LIN {X 0,Y 419.941,Z 601.82,A -85,B 0,C 180,E1 -10275.874,E2 -10275.874} C_VEL
LIN {X 0,Y 423.055,Z 612.363,A -85,B 0,C 180,E1 -10276.249,E2 -10276.249} C_VEL
LIN {X 0,Y 424.407,Z 618.673,A -85,B 0,C 180,E1 -10276.443,E2 -10276.443} C_VEL
LIN {X 0,Y 422.961,Z 707.954,A -85,B 0,C 180,E1 -10278.121,E2 -10278.121} C_VEL
LIN {X 0,Y 422.595,Z 721.713,A -85,B 0,C 180,E1 -10278.586,E2 -10278.586} C_VEL
LIN {X 0,Y 422.096,Z 733.741,A -85,B 0,C 180,E1 -10279.179,E2 -10279.179} C_VEL
LIN {X 0,Y 421.512,Z 745.803,A -85,B 0,C 180,E1 -10279.987,E2 -10279.987} C_VEL
LIN {X 0,Y 420.851,Z 757.025,A -85,B 0,C 180,E1 -10280.949,E2 -10280.949} C_VEL
LIN {X 0,Y 420.101,Z 766.764,A -85,B 0,C 180,E1 -10281.982,E2 -10281.982} C_VEL
LIN {X 0,Y 419.384,Z 776.447,A -85,B 0,C 180,E1 -10283.26,E2 -10283.26} C_VEL
LIN {X 0,Y 418.78,Z 784.344,A -85,B 0,C 180,E1 -10284.542,E2 -10284.542} C_VEL
LIN {X 0,Y 418.327,Z 791.168,A -85,B 0,C 180,E1 -10285.9,E2 -10285.9} C_VEL
LIN {X 0,Y 417.852,Z 797.772,A -85,B 0,C 180,E1 -10287.55,E2 -10287.55} C_VEL
LIN {X 0,Y 417.506,Z 802.788,A -85,B 0,C 180,E1 -10289.22,E2 -10289.22} C_VEL
LIN {X 0,Y 417.277,Z 806.247,A -85,B 0,C 180,E1 -10290.802,E2 -10290.802} C_VEL
LIN {X 0,Y 417.079,Z 808.819,A -85,B 0,C 180,E1 -10292.63,E2 -10292.63} C_VEL
LIN {X 0,Y 416.972,Z 809.86,A -85,B 0,C 180,E1 -10294.324,E2 -10294.324} C_VEL
LIN {X 0,Y 417.022,Z 809.583,A -85,B 0,C 180,E1 -10296.146,E2 -10296.146} C_VEL
LIN {X 0,Y 417.033,Z 808.324,A -85,B 0,C 180,E1 -10297.624,E2 -10297.624} C_VEL
LIN {X 0,Y 417.228,Z 805.887,A -85,B 0,C 180,E1 -10299.211,E2 -10299.211} C_VEL
LIN {X 0,Y 417.434,Z 802.41,A -85,B 0,C 180,E1 -10300.747,E2 -10300.747} C_VEL
LIN {X 0,Y 417.657,Z 797.653,A -85,B 0,C 180,E1 -10302.306,E2 -10302.306} C_VEL
LIN {X 0,Y 418.108,Z 791.143,A -85,B 0,C 180,E1 -10303.936,E2 -10303.936} C_VEL
LIN {X 0,Y 418.574,Z 784.013,A -85,B 0,C 180,E1 -10305.349,E2 -10305.349} C_VEL
LIN {X 0,Y 419.196,Z 775.516,A -85,B 0,C 180,E1 -10306.712,E2 -10306.712} C_VEL
LIN {X 0,Y 419.844,Z 765.863,A -85,B 0,C 180,E1 -10307.967,E2 -10307.967} C_VEL
LIN {X 0,Y 420.512,Z 755.212,A -85,B 0,C 180,E1 -10309.076,E2 -10309.076} C_VEL
LIN {X 0,Y 421.141,Z 744.253,A -85,B 0,C 180,E1 -10309.991,E2 -10309.991} C_VEL
LIN {X 0,Y 421.739,Z 733.285,A -85,B 0,C 180,E1 -10310.712,E2 -10310.712} C_VEL
LIN {X 0,Y 422.186,Z 720.348,A -85,B 0,C 180,E1 -10311.348,E2 -10311.348} C_VEL
LIN {X 0,Y 422.524,Z 707.087,A -85,B 0,C 180,E1 -10311.789,E2 -10311.789} C_VEL
LIN {X 0,Y 423.711,Z 617.543,A -85,B 0,C 180,E1 -10313.442,E2 -10313.442} C_VEL
LIN {X 0,Y 420.089,Z 601.796,A -85,B 0,C 180,E1 -10313.898,E2 -10313.898} C_VEL
LIN {X 0,Y 419.451,Z 599.695,A -85,B 0,C 180,E1 -10313.985,E2 -10313.985} C_VEL
LIN {X 0,Y 418.293,Z 593.383,A -85,B 0,C 180,E1 -10315.671,E2 -10315.671} C_VEL
LIN {X 0,Y 418.23,Z 593.385,A -85,B 0,C 180,E1 -10319.157,E2 -10319.157} C_VEL
LIN {X 0,Y 418.288,Z 593.383,A -85,B 0,C 180,E1 -10321.938,E2 -10321.938} C_VEL
LIN {X 0,Y 418.276,Z 593.378,A -85,B 0,C 180,E1 -10323.348,E2 -10323.348} C_VEL
LIN {X 0,Y 417.581,Z 593.471,A -85,B 0,C 180,E1 -10324.151,E2 -10324.151} C_VEL
LIN {X 0,Y 414.714,Z 593.823,A -85,B 0,C 180,E1 -10325.457,E2 -10325.457} C_VEL
LIN {X 0,Y 412.306,Z 594.125,A -85,B 0,C 180,E1 -10326.511,E2 -10326.511} C_VEL
LIN {X 0,Y 411.279,Z 594.25,A -85,B 0,C 180,E1 -10327.325,E2 -10327.325} C_VEL
LIN {X 0,Y 411.198,Z 594.261,A -85,B 0,C 180,E1 -10327.601,E2 -10327.601} C_VEL
LIN {X 0,Y 411.234,Z 594.255,A -85,B 0,C 180,E1 -10331.053,E2 -10331.053} C_VEL
LIN {X 0,Y 411.254,Z 594.259,A -85,B 0,C 180,E1 -10334.133,E2 -10334.133} C_VEL
LIN {X 0,Y 411.314,Z 594.245,A -85,B 0,C 180,E1 -10337.167,E2 -10337.167} C_VEL
LIN {X 0,Y 411.308,Z 594.251,A -85,B 0,C 180,E1 -10340.163,E2 -10340.163} C_VEL
LIN {X 0,Y 411.461,Z 594.228,A -85,B 0,C 180,E1 -10343.134,E2 -10343.134} C_VEL
LIN {X 0,Y 411.312,Z 594.247,A -85,B 0,C 180,E1 -10345.1,E2 -10345.1} C_VEL
LIN {X 0,Y 411.515,Z 594.222,A -85,B 0,C 180,E1 -10348.044,E2 -10348.044} C_VEL
LIN {X 0,Y 411.642,Z 594.206,A -85,B 0,C 180,E1 -10350.001,E2 -10350.001} C_VEL
LIN {X 0,Y 411.468,Z 594.23,A -85,B 0,C 180,E1 -10352.938,E2 -10352.938} C_VEL
LIN {X 0,Y 411.463,Z 594.232,A -85,B 0,C 180,E1 -10356.868,E2 -10356.868} C_VEL
LIN {X 0,Y 411.296,Z 594.248,A -85,B 0,C 180,E1 -10359.84,E2 -10359.84} C_VEL
LIN {X 0,Y 411.308,Z 594.25,A -85,B 0,C 180,E1 -10363.105,E2 -10363.105} C_VEL
LIN {X 0,Y 411.266,Z 594.259,A -85,B 0,C 180,E1 -10366.87,E2 -10366.87} C_VEL
LIN {X 0,Y 411.234,Z 594.255,A -85,B 0,C 180,E1 -10369.988,E2 -10369.988} C_VEL
LIN {X 0,Y 411.206,Z 594.264,A -85,B 0,C 180,E1 -10373.148,E2 -10373.148} C_VEL
LIN {X 0,Y 411.241,Z 594.255,A -85,B 0,C 180,E1 -10376.382,E2 -10376.382} C_VEL
LIN {X 0,Y 411.204,Z 594.26,A -85,B 0,C 180,E1 -10379.713,E2 -10379.713} C_VEL
LIN {X 0,Y 411.21,Z 594.266,A -85,B 0,C 180,E1 -10383.156,E2 -10383.156} C_VEL
LIN {X 0,Y 411.197,Z 594.261,A -85,B 0,C 180,E1 -10386.553,E2 -10386.553} C_VEL
LIN {X 0,Y 411.219,Z 594.26,A -85,B 0,C 180,E1 -10389.729,E2 -10389.729} C_VEL
LIN {X 0,Y 411.177,Z 594.268,A -85,B 0,C 180,E1 -10393.134,E2 -10393.134} C_VEL
LIN {X 0,Y 411.172,Z 594.265,A -85,B 0,C 180,E1 -10395.882,E2 -10395.882} C_VEL
LIN {X 0,Y 411.167,Z 594.264,A -85,B 0,C 180,E1 -10398.772,E2 -10398.772} C_VEL
LIN {X 0,Y 411.196,Z 594.262,A -85,B 0,C 180,E1 -10402.027,E2 -10402.027} C_VEL
LIN {X 0,Y 411.211,Z 594.265,A -85,B 0,C 180,E1 -10405.667,E2 -10405.667} C_VEL
LIN {X 0,Y 411.194,Z 594.262,A -85,B 0,C 180,E1 -10409.153,E2 -10409.153} C_VEL
LIN {X 0,Y 411.264,Z 594.252,A -85,B 0,C 180,E1 -10412.523,E2 -10412.523} C_VEL
LIN {X 0,Y 411.225,Z 594.264,A -85,B 0,C 180,E1 -10415.785,E2 -10415.785} C_VEL
LIN {X 0,Y 411.201,Z 594.26,A -85,B 0,C 180,E1 -10418.966,E2 -10418.966} C_VEL
LIN {X 0,Y 411.256,Z 594.257,A -85,B 0,C 180,E1 -10422.085,E2 -10422.085} C_VEL
LIN {X 0,Y 411.265,Z 594.252,A -85,B 0,C 180,E1 -10425.148,E2 -10425.148} C_VEL
LIN {X 0,Y 411.288,Z 594.254,A -85,B 0,C 180,E1 -10428.168,E2 -10428.168} C_VEL
LIN {X 0,Y 411.446,Z 594.235,A -85,B 0,C 180,E1 -10432.189,E2 -10432.189} C_VEL
LIN {X 0,Y 411.477,Z 594.232,A -85,B 0,C 180,E1 -10434.118,E2 -10434.118} C_VEL
LIN {X 0,Y 411.517,Z 594.226,A -85,B 0,C 180,E1 -10438.043,E2 -10438.043} C_VEL
LIN {X 0,Y 411.646,Z 594.209,A -85,B 0,C 180,E1 -10440,E2 -10440} C_VEL
LIN {X 0,Y 411.463,Z 594.227,A -85,B 0,C 180,E1 -10442.937,E2 -10442.937} C_VEL
LIN {X 0,Y 411.462,Z 594.229,A -85,B 0,C 180,E1 -10446.867,E2 -10446.867} C_VEL
LIN {X 0,Y 411.298,Z 594.249,A -85,B 0,C 180,E1 -10449.839,E2 -10449.839} C_VEL
LIN {X 0,Y 411.311,Z 594.246,A -85,B 0,C 180,E1 -10453.104,E2 -10453.104} C_VEL
LIN {X 0,Y 411.263,Z 594.255,A -85,B 0,C 180,E1 -10456.889,E2 -10456.889} C_VEL
LIN {X 0,Y 411.236,Z 594.256,A -85,B 0,C 180,E1 -10459.987,E2 -10459.987} C_VEL
LIN {X 0,Y 411.202,Z 594.261,A -85,B 0,C 180,E1 -10463.148,E2 -10463.148} C_VEL
LIN {X 0,Y 411.243,Z 594.258,A -85,B 0,C 180,E1 -10466.381,E2 -10466.381} C_VEL
LIN {X 0,Y 411.206,Z 594.259,A -85,B 0,C 180,E1 -10469.712,E2 -10469.712} C_VEL
LIN {X 0,Y 411.212,Z 594.261,A -85,B 0,C 180,E1 -10473.156,E2 -10473.156} C_VEL
LIN {X 0,Y 411.198,Z 594.264,A -85,B 0,C 180,E1 -10476.552,E2 -10476.552} C_VEL
LIN {X 0,Y 411.216,Z 594.258,A -85,B 0,C 180,E1 -10479.727,E2 -10479.727} C_VEL
LIN {X 0,Y 411.179,Z 594.268,A -85,B 0,C 180,E1 -10483.133,E2 -10483.133} C_VEL
LIN {X 0,Y 411.173,Z 594.263,A -85,B 0,C 180,E1 -10485.881,E2 -10485.881} C_VEL
LIN {X 0,Y 411.169,Z 594.267,A -85,B 0,C 180,E1 -10488.771,E2 -10488.771} C_VEL
LIN {X 0,Y 411.21,Z 594.259,A -85,B 0,C 180,E1 -10491.831,E2 -10491.831} C_VEL
LIN {X 0,Y 411.216,Z 594.264,A -85,B 0,C 180,E1 -10495.121,E2 -10495.121} C_VEL
LIN {X 0,Y 411.171,Z 594.266,A -85,B 0,C 180,E1 -10498.002,E2 -10498.002} C_VEL
LIN {X 0,Y 411.261,Z 594.413,A -85,B 0,C 180,E1 -10500.79,E2 -10500.79} C_VEL
LIN {X 0,Y 414.087,Z 607.419,A -85,B 0,C 180,E1 -10503.542,E2 -10503.542} C_VEL
LIN {X 0,Y 414.89,Z 613.069,A -85,B 0,C 180,E1 -10504.687,E2 -10504.687} C_VEL
LIN {X 0,Y 413.836,Z 628.092,A -85,B 0,C 180,E1 -10507.535,E2 -10507.535} C_VEL
LIN {X 0,Y 412.832,Z 643.304,A -85,B 0,C 180,E1 -10510.378,E2 -10510.378} C_VEL
LIN {X 0,Y 412.697,Z 645.191,A -85,B 0,C 180,E1 -10510.729,E2 -10510.729} C_VEL
LIN {X 0,Y 416.641,Z 674.102,A -85,B 0,C 180,E1 -10511.462,E2 -10511.462} C_VEL
LIN {X 0,Y 415.489,Z 754.532,A -85,B 0,C 180,E1 -10512.971,E2 -10512.971} C_VEL
LIN {X 0,Y 414.975,Z 768.128,A -85,B 0,C 180,E1 -10513.424,E2 -10513.424} C_VEL
LIN {X 0,Y 414.351,Z 779.945,A -85,B 0,C 180,E1 -10514,E2 -10514} C_VEL
LIN {X 0,Y 413.654,Z 791.204,A -85,B 0,C 180,E1 -10514.73,E2 -10514.73} C_VEL
LIN {X 0,Y 412.918,Z 802.904,A -85,B 0,C 180,E1 -10515.712,E2 -10515.712} C_VEL
LIN {X 0,Y 412.199,Z 813.634,A -85,B 0,C 180,E1 -10516.839,E2 -10516.839} C_VEL
LIN {X 0,Y 411.651,Z 822.069,A -85,B 0,C 180,E1 -10517.927,E2 -10517.927} C_VEL
LIN {X 0,Y 411.016,Z 830.01,A -85,B 0,C 180,E1 -10519.158,E2 -10519.158} C_VEL
LIN {X 0,Y 410.584,Z 837.764,A -85,B 0,C 180,E1 -10520.64,E2 -10520.64} C_VEL
LIN {X 0,Y 410.274,Z 843.987,A -85,B 0,C 180,E1 -10522.122,E2 -10522.122} C_VEL
LIN {X 0,Y 410.107,Z 849.181,A -85,B 0,C 180,E1 -10523.695,E2 -10523.695} C_VEL
LIN {X 0,Y 410.079,Z 852.686,A -85,B 0,C 180,E1 -10525.083,E2 -10525.083} C_VEL
LIN {X 0,Y 409.971,Z 854.618,A -85,B 0,C 180,E1 -10526.067,E2 -10526.067} C_VEL
LIN {X 0,Y 410.053,Z 856.108,A -85,B 0,C 180,E1 -10527.052,E2 -10527.052} C_VEL
LIN {X 0,Y 410.059,Z 857.14,A -85,B 0,C 180,E1 -10528.035,E2 -10528.035} C_VEL
LIN {X 0,Y 410.027,Z 857.768,A -85,B 0,C 180,E1 -10529.017,E2 -10529.017} C_VEL
LIN {X 0,Y 410.033,Z 857.996,A -85,B 0,C 180,E1 -10529.999,E2 -10529.999} C_VEL
LIN {X 0,Y 410.027,Z 857.792,A -85,B 0,C 180,E1 -10530.981,E2 -10530.981} C_VEL
LIN {X 0,Y 410.06,Z 857.161,A -85,B 0,C 180,E1 -10531.963,E2 -10531.963} C_VEL
LIN {X 0,Y 410.055,Z 856.128,A -85,B 0,C 180,E1 -10532.946,E2 -10532.946} C_VEL
LIN {X 0,Y 409.969,Z 854.68,A -85,B 0,C 180,E1 -10533.931,E2 -10533.931} C_VEL
LIN {X 0,Y 410.042,Z 851.651,A -85,B 0,C 180,E1 -10535.408,E2 -10535.408} C_VEL
LIN {X 0,Y 410.163,Z 847.56,A -85,B 0,C 180,E1 -10536.888,E2 -10536.888} C_VEL
LIN {X 0,Y 410.411,Z 841.281,A -85,B 0,C 180,E1 -10538.616,E2 -10538.616} C_VEL
LIN {X 0,Y 410.816,Z 834.425,A -85,B 0,C 180,E1 -10540.098,E2 -10540.098} C_VEL
LIN {X 0,Y 411.389,Z 825.935,A -85,B 0,C 180,E1 -10541.579,E2 -10541.579} C_VEL
LIN {X 0,Y 411.949,Z 817.225,A -85,B 0,C 180,E1 -10542.813,E2 -10542.813} C_VEL
LIN {X 0,Y 412.72,Z 806.761,A -85,B 0,C 180,E1 -10544.017,E2 -10544.017} C_VEL
LIN {X 0,Y 413.498,Z 795.956,A -85,B 0,C 180,E1 -10545.021,E2 -10545.021} C_VEL
LIN {X 0,Y 414.343,Z 784.371,A -85,B 0,C 180,E1 -10545.872,E2 -10545.872} C_VEL
LIN {X 0,Y 415.045,Z 771.148,A -85,B 0,C 180,E1 -10546.602,E2 -10546.602} C_VEL
LIN {X 0,Y 415.738,Z 757.929,A -85,B 0,C 180,E1 -10547.111,E2 -10547.111} C_VEL
LIN {X 0,Y 416.035,Z 743.572,A -85,B 0,C 180,E1 -10547.447,E2 -10547.447} C_VEL
LIN {X 0,Y 417.035,Z 672.509,A -85,B 0,C 180,E1 -10548.788,E2 -10548.788} C_VEL
LIN {X 0,Y 413.245,Z 645.793,A -85,B 0,C 180,E1 -10549.525,E2 -10549.525} C_VEL
LIN {X 0,Y 412.815,Z 643.284,A -85,B 0,C 180,E1 -10549.621,E2 -10549.621} C_VEL
LIN {X 0,Y 414.034,Z 625.579,A -85,B 0,C 180,E1 -10552.979,E2 -10552.979} C_VEL
LIN {X 0,Y 414.946,Z 612.192,A -85,B 0,C 180,E1 -10555.573,E2 -10555.573} C_VEL
LIN {X 0,Y 413.027,Z 602.03,A -85,B 0,C 180,E1 -10557.77,E2 -10557.77} C_VEL
LIN {X 0,Y 411.226,Z 594.263,A -85,B 0,C 180,E1 -10559.539,E2 -10559.539} C_VEL
LIN {X 0,Y 411.203,Z 594.266,A -85,B 0,C 180,E1 -10563.155,E2 -10563.155} C_VEL
LIN {X 0,Y 411.193,Z 594.268,A -85,B 0,C 180,E1 -10566.552,E2 -10566.552} C_VEL
LIN {X 0,Y 411.224,Z 594.262,A -85,B 0,C 180,E1 -10569.729,E2 -10569.729} C_VEL
LIN {X 0,Y 411.173,Z 594.269,A -85,B 0,C 180,E1 -10573.132,E2 -10573.132} C_VEL
LIN {X 0,Y 411.231,Z 594.261,A -85,B 0,C 180,E1 -10575.87,E2 -10575.87} C_VEL
LIN {X 0,Y 411.205,Z 594.263,A -85,B 0,C 180,E1 -10578.763,E2 -10578.763} C_VEL
LIN {X 0,Y 411.199,Z 594.263,A -85,B 0,C 180,E1 -10582.027,E2 -10582.027} C_VEL
LIN {X 0,Y 411.2,Z 594.261,A -85,B 0,C 180,E1 -10585.666,E2 -10585.666} C_VEL
LIN {X 0,Y 411.194,Z 594.261,A -85,B 0,C 180,E1 -10589.153,E2 -10589.153} C_VEL
LIN {X 0,Y 411.252,Z 594.258,A -85,B 0,C 180,E1 -10592.522,E2 -10592.522} C_VEL
LIN {X 0,Y 411.219,Z 594.259,A -85,B 0,C 180,E1 -10595.784,E2 -10595.784} C_VEL
LIN {X 0,Y 411.189,Z 594.261,A -85,B 0,C 180,E1 -10598.965,E2 -10598.965} C_VEL
LIN {X 0,Y 411.245,Z 594.259,A -85,B 0,C 180,E1 -10602.084,E2 -10602.084} C_VEL
LIN {X 0,Y 411.254,Z 594.253,A -85,B 0,C 180,E1 -10605.147,E2 -10605.147} C_VEL
LIN {X 0,Y 411.291,Z 594.252,A -85,B 0,C 180,E1 -10608.167,E2 -10608.167} C_VEL
LIN {X 0,Y 411.473,Z 594.232,A -85,B 0,C 180,E1 -10612.146,E2 -10612.146} C_VEL
LIN {X 0,Y 411.467,Z 594.233,A -85,B 0,C 180,E1 -10614.118,E2 -10614.118} C_VEL
LIN {X 0,Y 411.506,Z 594.228,A -85,B 0,C 180,E1 -10618.042,E2 -10618.042} C_VEL
LIN {X 0,Y 411.635,Z 594.212,A -85,B 0,C 180,E1 -10620,E2 -10620} C_VEL
LIN {X 0,Y 411.46,Z 594.232,A -85,B 0,C 180,E1 -10622.937,E2 -10622.937} C_VEL
LIN {X 0,Y 411.45,Z 594.234,A -85,B 0,C 180,E1 -10626.608,E2 -10626.608} C_VEL
LIN {X 0,Y 411.349,Z 594.247,A -85,B 0,C 180,E1 -10628.845,E2 -10628.845} C_VEL
LIN {X 0,Y 411.29,Z 594.255,A -85,B 0,C 180,E1 -10631.832,E2 -10631.832} C_VEL
LIN {X 0,Y 411.347,Z 594.455,A -85,B 0,C 180,E1 -10633.257,E2 -10633.257} C_VEL
LIN {X 0,Y 412.864,Z 602.289,A -85,B 0,C 180,E1 -10635.488,E2 -10635.488} C_VEL
LIN {X 0,Y 416.193,Z 612.686,A -85,B 0,C 180,E1 -10635.889,E2 -10635.889} C_VEL
LIN {X 0,Y 417.739,Z 620.471,A -85,B 0,C 180,E1 -10636.134,E2 -10636.134} C_VEL
LIN {X 0,Y 416.229,Z 708.435,A -85,B 0,C 180,E1 -10637.821,E2 -10637.821} C_VEL
LIN {X 0,Y 415.844,Z 721.956,A -85,B 0,C 180,E1 -10638.283,E2 -10638.283} C_VEL
LIN {X 0,Y 415.29,Z 735.058,A -85,B 0,C 180,E1 -10638.948,E2 -10638.948} C_VEL
LIN {X 0,Y 414.658,Z 747.51,A -85,B 0,C 180,E1 -10639.815,E2 -10639.815} C_VEL
LIN {X 0,Y 413.929,Z 758.735,A -85,B 0,C 180,E1 -10640.815,E2 -10640.815} C_VEL
LIN {X 0,Y 413.092,Z 769.11,A -85,B 0,C 180,E1 -10641.98,E2 -10641.98} C_VEL
LIN {X 0,Y 412.325,Z 778.874,A -85,B 0,C 180,E1 -10643.346,E2 -10643.346} C_VEL
LIN {X 0,Y 411.652,Z 786.824,A -85,B 0,C 180,E1 -10644.726,E2 -10644.726} C_VEL
LIN {X 0,Y 411.147,Z 794.377,A -85,B 0,C 180,E1 -10646.387,E2 -10646.387} C_VEL
LIN {X 0,Y 410.697,Z 800.355,A -85,B 0,C 180,E1 -10648.073,E2 -10648.073} C_VEL
LIN {X 0,Y 410.369,Z 804.818,A -85,B 0,C 180,E1 -10649.779,E2 -10649.779} C_VEL
LIN {X 0,Y 410.185,Z 807.283,A -85,B 0,C 180,E1 -10651.056,E2 -10651.056} C_VEL
LIN {X 0,Y 409.98,Z 809.49,A -85,B 0,C 180,E1 -10652.865,E2 -10652.865} C_VEL
LIN {X 0,Y 409.888,Z 810.32,A -85,B 0,C 180,E1 -10654.615,E2 -10654.615} C_VEL
LIN {X 0,Y 409.929,Z 809.907,A -85,B 0,C 180,E1 -10656.316,E2 -10656.316} C_VEL
LIN {X 0,Y 409.995,Z 808.179,A -85,B 0,C 180,E1 -10658.105,E2 -10658.105} C_VEL
LIN {X 0,Y 410.28,Z 804.688,A -85,B 0,C 180,E1 -10660.041,E2 -10660.041} C_VEL
LIN {X 0,Y 410.471,Z 801.03,A -85,B 0,C 180,E1 -10661.462,E2 -10661.462} C_VEL
LIN {X 0,Y 410.803,Z 795.209,A -85,B 0,C 180,E1 -10663.182,E2 -10663.182} C_VEL
LIN {X 0,Y 411.349,Z 788.305,A -85,B 0,C 180,E1 -10664.748,E2 -10664.748} C_VEL
LIN {X 0,Y 411.793,Z 780.664,A -85,B 0,C 180,E1 -10666.143,E2 -10666.143} C_VEL
LIN {X 0,Y 412.522,Z 771.747,A -85,B 0,C 180,E1 -10667.463,E2 -10667.463} C_VEL
LIN {X 0,Y 413.204,Z 762.025,A -85,B 0,C 180,E1 -10668.634,E2 -10668.634} C_VEL
LIN {X 0,Y 413.878,Z 751.635,A -85,B 0,C 180,E1 -10669.642,E2 -10669.642} C_VEL
LIN {X 0,Y 414.506,Z 740.413,A -85,B 0,C 180,E1 -10670.513,E2 -10670.513} C_VEL
LIN {X 0,Y 415.142,Z 727.922,A -85,B 0,C 180,E1 -10671.259,E2 -10671.259} C_VEL
LIN {X 0,Y 415.482,Z 714.834,A -85,B 0,C 180,E1 -10671.817,E2 -10671.817} C_VEL
LIN {X 0,Y 415.832,Z 701.375,A -85,B 0,C 180,E1 -10672.177,E2 -10672.177} C_VEL
LIN {X 0,Y 416.911,Z 618.483,A -85,B 0,C 180,E1 -10673.714,E2 -10673.714} C_VEL
LIN {X 0,Y 413.739,Z 604.516,A -85,B 0,C 180,E1 -10674.125,E2 -10674.125} C_VEL
LIN {X 0,Y 412.346,Z 600.121,A -85,B 0,C 180,E1 -10674.286,E2 -10674.286} C_VEL
LIN {X 0,Y 411.247,Z 594.26,A -85,B 0,C 180,E1 -10675.894,E2 -10675.894} C_VEL
LIN {X 0,Y 411.185,Z 594.262,A -85,B 0,C 180,E1 -10679.154,E2 -10679.154} C_VEL
LIN {X 0,Y 411.255,Z 594.255,A -85,B 0,C 180,E1 -10682.523,E2 -10682.523} C_VEL
LIN {X 0,Y 411.225,Z 594.26,A -85,B 0,C 180,E1 -10685.786,E2 -10685.786} C_VEL
LIN {X 0,Y 411.198,Z 594.261,A -85,B 0,C 180,E1 -10687.601,E2 -10687.601} C_VEL
LIN {X 0,Y 410.548,Z 594.349,A -85,B 0,C 180,E1 -10688.419,E2 -10688.419} C_VEL
LIN {X 0,Y 407.736,Z 594.701,A -85,B 0,C 180,E1 -10689.748,E2 -10689.748} C_VEL
LIN {X 0,Y 405.341,Z 594.997,A -85,B 0,C 180,E1 -10690.822,E2 -10690.822} C_VEL
LIN {X 0,Y 404.295,Z 595.122,A -85,B 0,C 180,E1 -10691.651,E2 -10691.651} C_VEL
LIN {X 0,Y 404.202,Z 595.132,A -85,B 0,C 180,E1 -10691.932,E2 -10691.932} C_VEL
LIN {X 0,Y 404.207,Z 595.132,A -85,B 0,C 180,E1 -10694.883,E2 -10694.883} C_VEL
LIN {X 0,Y 404.27,Z 595.126,A -85,B 0,C 180,E1 -10697.96,E2 -10697.96} C_VEL
LIN {X 0,Y 404.433,Z 595.106,A -85,B 0,C 180,E1 -10702.101,E2 -10702.101} C_VEL
LIN {X 0,Y 404.424,Z 595.106,A -85,B 0,C 180,E1 -10704.016,E2 -10704.016} C_VEL
LIN {X 0,Y 404.484,Z 595.098,A -85,B 0,C 180,E1 -10708.01,E2 -10708.01} C_VEL
LIN {X 0,Y 404.611,Z 595.082,A -85,B 0,C 180,E1 -10710.001,E2 -10710.001} C_VEL
LIN {X 0,Y 404.425,Z 595.107,A -85,B 0,C 180,E1 -10712.989,E2 -10712.989} C_VEL
LIN {X 0,Y 404.414,Z 595.109,A -85,B 0,C 180,E1 -10716.988,E2 -10716.988} C_VEL
LIN {X 0,Y 404.261,Z 595.125,A -85,B 0,C 180,E1 -10720.013,E2 -10720.013} C_VEL
LIN {X 0,Y 404.269,Z 595.126,A -85,B 0,C 180,E1 -10723.212,E2 -10723.212} C_VEL
LIN {X 0,Y 404.219,Z 595.135,A -85,B 0,C 180,E1 -10727.008,E2 -10727.008} C_VEL
LIN {X 0,Y 404.167,Z 595.137,A -85,B 0,C 180,E1 -10730.352,E2 -10730.352} C_VEL
LIN {X 0,Y 404.173,Z 595.136,A -85,B 0,C 180,E1 -10733.575,E2 -10733.575} C_VEL
LIN {X 0,Y 404.187,Z 595.134,A -85,B 0,C 180,E1 -10735.767,E2 -10735.767} C_VEL
LIN {X 0,Y 404.199,Z 595.132,A -85,B 0,C 180,E1 -10738,E2 -10738} C_VEL
LIN {X 0,Y 404.143,Z 595.141,A -85,B 0,C 180,E1 -10741.559,E2 -10741.559} C_VEL
LIN {X 0,Y 404.189,Z 595.138,A -85,B 0,C 180,E1 -10745.017,E2 -10745.017} C_VEL
LIN {X 0,Y 404.16,Z 595.139,A -85,B 0,C 180,E1 -10748.757,E2 -10748.757} C_VEL
LIN {X 0,Y 404.127,Z 595.145,A -85,B 0,C 180,E1 -10751.6,E2 -10751.6} C_VEL
LIN {X 0,Y 404.149,Z 595.138,A -85,B 0,C 180,E1 -10754.523,E2 -10754.523} C_VEL
LIN {X 0,Y 404.14,Z 595.145,A -85,B 0,C 180,E1 -10757.296,E2 -10757.296} C_VEL
LIN {X 0,Y 404.173,Z 595.137,A -85,B 0,C 180,E1 -10759.956,E2 -10759.956} C_VEL
LIN {X 0,Y 404.14,Z 595.142,A -85,B 0,C 180,E1 -10763.126,E2 -10763.126} C_VEL
LIN {X 0,Y 404.15,Z 595.139,A -85,B 0,C 180,E1 -10766.188,E2 -10766.188} C_VEL
LIN {X 0,Y 404.15,Z 595.144,A -85,B 0,C 180,E1 -10769.715,E2 -10769.715} C_VEL
LIN {X 0,Y 404.2,Z 595.133,A -85,B 0,C 180,E1 -10773.123,E2 -10773.123} C_VEL
LIN {X 0,Y 404.179,Z 595.137,A -85,B 0,C 180,E1 -10775.335,E2 -10775.335} C_VEL
LIN {X 0,Y 404.143,Z 595.139,A -85,B 0,C 180,E1 -10778.581,E2 -10778.581} C_VEL
LIN {X 0,Y 404.214,Z 595.136,A -85,B 0,C 180,E1 -10781.762,E2 -10781.762} C_VEL
LIN {X 0,Y 404.211,Z 595.13,A -85,B 0,C 180,E1 -10784.882,E2 -10784.882} C_VEL
LIN {X 0,Y 404.261,Z 595.132,A -85,B 0,C 180,E1 -10787.959,E2 -10787.959} C_VEL
LIN {X 0,Y 404.411,Z 595.112,A -85,B 0,C 180,E1 -10792.129,E2 -10792.129} C_VEL
LIN {X 0,Y 404.426,Z 595.11,A -85,B 0,C 180,E1 -10794.015,E2 -10794.015} C_VEL
LIN {X 0,Y 404.486,Z 595.102,A -85,B 0,C 180,E1 -10798.009,E2 -10798.009} C_VEL
LIN {X 0,Y 404.615,Z 595.085,A -85,B 0,C 180,E1 -10800,E2 -10800} C_VEL
LIN {X 0,Y 404.421,Z 595.104,A -85,B 0,C 180,E1 -10802.989,E2 -10802.989} C_VEL
LIN {X 0,Y 404.429,Z 595.107,A -85,B 0,C 180,E1 -10805.985,E2 -10805.985} C_VEL
LIN {X 0,Y 404.297,Z 595.12,A -85,B 0,C 180,E1 -10809.001,E2 -10809.001} C_VEL
LIN {X 0,Y 404.262,Z 595.127,A -85,B 0,C 180,E1 -10812.042,E2 -10812.042} C_VEL
LIN {X 0,Y 404.212,Z 595.131,A -85,B 0,C 180,E1 -10815.118,E2 -10815.118} C_VEL
LIN {X 0,Y 404.21,Z 595.134,A -85,B 0,C 180,E1 -10818.238,E2 -10818.238} C_VEL
LIN {X 0,Y 404.144,Z 595.139,A -85,B 0,C 180,E1 -10821.419,E2 -10821.419} C_VEL
LIN {X 0,Y 404.181,Z 595.141,A -85,B 0,C 180,E1 -10824.666,E2 -10824.666} C_VEL
LIN {X 0,Y 404.201,Z 595.132,A -85,B 0,C 180,E1 -10827.999,E2 -10827.999} C_VEL
LIN {X 0,Y 404.145,Z 595.139,A -85,B 0,C 180,E1 -10831.558,E2 -10831.558} C_VEL
LIN {X 0,Y 404.19,Z 595.138,A -85,B 0,C 180,E1 -10835.016,E2 -10835.016} C_VEL
LIN {X 0,Y 404.158,Z 595.143,A -85,B 0,C 180,E1 -10838.757,E2 -10838.757} C_VEL
LIN {X 0,Y 404.128,Z 595.141,A -85,B 0,C 180,E1 -10841.599,E2 -10841.599} C_VEL
LIN {X 0,Y 404.151,Z 595.14,A -85,B 0,C 180,E1 -10844.522,E2 -10844.522} C_VEL
LIN {X 0,Y 404.142,Z 595.143,A -85,B 0,C 180,E1 -10847.295,E2 -10847.295} C_VEL
LIN {X 0,Y 404.174,Z 595.135,A -85,B 0,C 180,E1 -10849.955,E2 -10849.955} C_VEL
LIN {X 0,Y 404.142,Z 595.146,A -85,B 0,C 180,E1 -10853.124,E2 -10853.124} C_VEL
LIN {X 0,Y 404.15,Z 595.141,A -85,B 0,C 180,E1 -10856.187,E2 -10856.187} C_VEL
LIN {X 0,Y 404.151,Z 595.143,A -85,B 0,C 180,E1 -10859.714,E2 -10859.714} C_VEL
LIN {X 0,Y 404.225,Z 595.308,A -85,B 0,C 180,E1 -10860.526,E2 -10860.526} C_VEL
LIN {X 0,Y 407.296,Z 609.706,A -85,B 0,C 180,E1 -10863.626,E2 -10863.626} C_VEL
LIN {X 0,Y 407.921,Z 615.249,A -85,B 0,C 180,E1 -10864.759,E2 -10864.759} C_VEL
LIN {X 0,Y 406.554,Z 633.071,A -85,B 0,C 180,E1 -10868.181,E2 -10868.181} C_VEL
LIN {X 0,Y 405.787,Z 645.051,A -85,B 0,C 180,E1 -10870.425,E2 -10870.425} C_VEL
LIN {X 0,Y 409.84,Z 674.732,A -85,B 0,C 180,E1 -10871.192,E2 -10871.192} C_VEL
LIN {X 0,Y 408.637,Z 754.065,A -85,B 0,C 180,E1 -10872.709,E2 -10872.709} C_VEL
LIN {X 0,Y 408.115,Z 767.669,A -85,B 0,C 180,E1 -10873.17,E2 -10873.17} C_VEL
LIN {X 0,Y 407.428,Z 780.048,A -85,B 0,C 180,E1 -10873.785,E2 -10873.785} C_VEL
LIN {X 0,Y 406.648,Z 791.962,A -85,B 0,C 180,E1 -10874.589,E2 -10874.589} C_VEL
LIN {X 0,Y 405.905,Z 803.449,A -85,B 0,C 180,E1 -10875.587,E2 -10875.587} C_VEL
LIN {X 0,Y 405.158,Z 814.19,A -85,B 0,C 180,E1 -10876.757,E2 -10876.757} C_VEL
LIN {X 0,Y 404.518,Z 823.139,A -85,B 0,C 180,E1 -10877.965,E2 -10877.965} C_VEL
LIN {X 0,Y 403.799,Z 832.193,A -85,B 0,C 180,E1 -10879.469,E2 -10879.469} C_VEL
LIN {X 0,Y 403.396,Z 839.482,A -85,B 0,C 180,E1 -10880.978,E2 -10880.978} C_VEL
LIN {X 0,Y 403.131,Z 845.276,A -85,B 0,C 180,E1 -10882.486,E2 -10882.486} C_VEL
LIN {X 0,Y 402.988,Z 849.823,A -85,B 0,C 180,E1 -10883.993,E2 -10883.993} C_VEL
LIN {X 0,Y 402.987,Z 852.216,A -85,B 0,C 180,E1 -10884.996,E2 -10884.996} C_VEL
LIN {X 0,Y 402.891,Z 854.16,A -85,B 0,C 180,E1 -10885.998,E2 -10885.998} C_VEL
LIN {X 0,Y 402.953,Z 855.666,A -85,B 0,C 180,E1 -10887,E2 -10887} C_VEL
LIN {X 0,Y 402.987,Z 856.709,A -85,B 0,C 180,E1 -10888,E2 -10888} C_VEL
LIN {X 0,Y 402.949,Z 857.342,A -85,B 0,C 180,E1 -10889,E2 -10889} C_VEL
LIN {X 0,Y 402.952,Z 857.577,A -85,B 0,C 180,E1 -10889.999,E2 -10889.999} C_VEL
LIN {X 0,Y 402.949,Z 857.386,A -85,B 0,C 180,E1 -10890.998,E2 -10890.998} C_VEL
LIN {X 0,Y 402.988,Z 856.76,A -85,B 0,C 180,E1 -10891.998,E2 -10891.998} C_VEL
LIN {X 0,Y 402.953,Z 855.727,A -85,B 0,C 180,E1 -10892.998,E2 -10892.998} C_VEL
LIN {X 0,Y 402.888,Z 854.283,A -85,B 0,C 180,E1 -10894,E2 -10894} C_VEL
LIN {X 0,Y 402.942,Z 851.259,A -85,B 0,C 180,E1 -10895.504,E2 -10895.504} C_VEL
LIN {X 0,Y 403.074,Z 847.173,A -85,B 0,C 180,E1 -10897.009,E2 -10897.009} C_VEL
LIN {X 0,Y 403.36,Z 840.903,A -85,B 0,C 180,E1 -10898.768,E2 -10898.768} C_VEL
LIN {X 0,Y 403.76,Z 834.065,A -85,B 0,C 180,E1 -10900.276,E2 -10900.276} C_VEL
LIN {X 0,Y 404.394,Z 825.603,A -85,B 0,C 180,E1 -10901.782,E2 -10901.782} C_VEL
LIN {X 0,Y 405.008,Z 816.94,A -85,B 0,C 180,E1 -10903.036,E2 -10903.036} C_VEL
LIN {X 0,Y 405.834,Z 806.267,A -85,B 0,C 180,E1 -10904.285,E2 -10904.285} C_VEL
LIN {X 0,Y 406.716,Z 794.283,A -85,B 0,C 180,E1 -10905.406,E2 -10905.406} C_VEL
LIN {X 0,Y 407.646,Z 782.249,A -85,B 0,C 180,E1 -10906.268,E2 -10906.268} C_VEL
LIN {X 0,Y 408.267,Z 771.108,A -85,B 0,C 180,E1 -10906.886,E2 -10906.886} C_VEL
LIN {X 0,Y 408.982,Z 758.072,A -85,B 0,C 180,E1 -10907.403,E2 -10907.403} C_VEL
LIN {X 0,Y 409.296,Z 744.251,A -85,B 0,C 180,E1 -10907.744,E2 -10907.744} C_VEL
LIN {X 0,Y 410.386,Z 673.481,A -85,B 0,C 180,E1 -10909.108,E2 -10909.108} C_VEL
LIN {X 0,Y 406.919,Z 648.533,A -85,B 0,C 180,E1 -10909.816,E2 -10909.816} C_VEL
LIN {X 0,Y 405.94,Z 642.849,A -85,B 0,C 180,E1 -10910.003,E2 -10910.003} C_VEL
LIN {X 0,Y 407.384,Z 623.495,A -85,B 0,C 180,E1 -10913.755,E2 -10913.755} C_VEL
LIN {X 0,Y 408.093,Z 614.661,A -85,B 0,C 180,E1 -10915.5,E2 -10915.5} C_VEL
LIN {X 0,Y 407.037,Z 607.973,A -85,B 0,C 180,E1 -10916.95,E2 -10916.95} C_VEL
LIN {X 0,Y 404.578,Z 596.93,A -85,B 0,C 180,E1 -10919.485,E2 -10919.485} C_VEL
LIN {X 0,Y 404.175,Z 595.142,A -85,B 0,C 180,E1 -10919.946,E2 -10919.946} C_VEL
LIN {X 0,Y 404.142,Z 595.144,A -85,B 0,C 180,E1 -10923.811,E2 -10923.811} C_VEL
LIN {X 0,Y 404.137,Z 595.146,A -85,B 0,C 180,E1 -10926.875,E2 -10926.875} C_VEL
LIN {X 0,Y 404.163,Z 595.144,A -85,B 0,C 180,E1 -10930.082,E2 -10930.082} C_VEL
LIN {X 0,Y 404.153,Z 595.144,A -85,B 0,C 180,E1 -10933.083,E2 -10933.083} C_VEL
LIN {X 0,Y 404.204,Z 595.137,A -85,B 0,C 180,E1 -10935.933,E2 -10935.933} C_VEL
LIN {X 0,Y 404.159,Z 595.141,A -85,B 0,C 180,E1 -10938.64,E2 -10938.64} C_VEL
LIN {X 0,Y 404.157,Z 595.138,A -85,B 0,C 180,E1 -10941.49,E2 -10941.49} C_VEL
LIN {X 0,Y 404.179,Z 595.137,A -85,B 0,C 180,E1 -10944.983,E2 -10944.983} C_VEL
LIN {X 0,Y 404.143,Z 595.14,A -85,B 0,C 180,E1 -10948.554,E2 -10948.554} C_VEL
LIN {X 0,Y 404.191,Z 595.132,A -85,B 0,C 180,E1 -10952,E2 -10952} C_VEL
LIN {X 0,Y 404.169,Z 595.136,A -85,B 0,C 180,E1 -10955.334,E2 -10955.334} C_VEL
LIN {X 0,Y 404.152,Z 595.142,A -85,B 0,C 180,E1 -10958.581,E2 -10958.581} C_VEL
LIN {X 0,Y 404.202,Z 595.135,A -85,B 0,C 180,E1 -10961.761,E2 -10961.761} C_VEL
LIN {X 0,Y 404.199,Z 595.132,A -85,B 0,C 180,E1 -10964.882,E2 -10964.882} C_VEL
LIN {X 0,Y 404.262,Z 595.126,A -85,B 0,C 180,E1 -10967.958,E2 -10967.958} C_VEL
LIN {X 0,Y 404.425,Z 595.11,A -85,B 0,C 180,E1 -10972.099,E2 -10972.099} C_VEL
LIN {X 0,Y 404.416,Z 595.111,A -85,B 0,C 180,E1 -10974.015,E2 -10974.015} C_VEL
LIN {X 0,Y 404.475,Z 595.104,A -85,B 0,C 180,E1 -10978.008,E2 -10978.008} C_VEL
LIN {X 0,Y 404.605,Z 595.088,A -85,B 0,C 180,E1 -10980,E2 -10980} C_VEL
LIN {X 0,Y 404.417,Z 595.109,A -85,B 0,C 180,E1 -10982.988,E2 -10982.988} C_VEL
LIN {X 0,Y 404.4,Z 595.112,A -85,B 0,C 180,E1 -10986.606,E2 -10986.606} C_VEL
LIN {X 0,Y 404.288,Z 595.126,A -85,B 0,C 180,E1 -10989.001,E2 -10989.001} C_VEL
LIN {X 0,Y 404.277,Z 595.132,A -85,B 0,C 180,E1 -10992.838,E2 -10992.838} C_VEL
LIN {X 0,Y 405.798,Z 602.861,A -85,B 0,C 180,E1 -10995.089,E2 -10995.089} C_VEL
LIN {X 0,Y 409.519,Z 613.62,A -85,B 0,C 180,E1 -10995.533,E2 -10995.533} C_VEL
LIN {X 0,Y 411.153,Z 621.227,A -85,B 0,C 180,E1 -10995.785,E2 -10995.785} C_VEL
LIN {X 0,Y 409.514,Z 708.92,A -85,B 0,C 180,E1 -10997.51,E2 -10997.51} C_VEL
LIN {X 0,Y 409.125,Z 722.369,A -85,B 0,C 180,E1 -10997.979,E2 -10997.979} C_VEL
LIN {X 0,Y 408.6,Z 734.232,A -85,B 0,C 180,E1 -10998.579,E2 -10998.579} C_VEL
LIN {X 0,Y 407.977,Z 745.841,A -85,B 0,C 180,E1 -10999.366,E2 -10999.366} C_VEL
LIN {X 0,Y 407.283,Z 756.715,A -85,B 0,C 180,E1 -11000.311,E2 -11000.311} C_VEL
LIN {X 0,Y 406.415,Z 767.072,A -85,B 0,C 180,E1 -11001.426,E2 -11001.426} C_VEL
LIN {X 0,Y 405.691,Z 776.203,A -85,B 0,C 180,E1 -11002.643,E2 -11002.643} C_VEL
LIN {X 0,Y 404.914,Z 784.853,A -85,B 0,C 180,E1 -11004.072,E2 -11004.072} C_VEL
LIN {X 0,Y 404.401,Z 791.204,A -85,B 0,C 180,E1 -11005.355,E2 -11005.355} C_VEL
LIN {X 0,Y 403.917,Z 797.381,A -85,B 0,C 180,E1 -11006.897,E2 -11006.897} C_VEL
LIN {X 0,Y 403.497,Z 802.739,A -85,B 0,C 180,E1 -11008.619,E2 -11008.619} C_VEL
LIN {X 0,Y 403.209,Z 806.655,A -85,B 0,C 180,E1 -11010.363,E2 -11010.363} C_VEL
LIN {X 0,Y 403.021,Z 808.54,A -85,B 0,C 180,E1 -11011.544,E2 -11011.544} C_VEL
LIN {X 0,Y 402.854,Z 810.166,A -85,B 0,C 180,E1 -11013.138,E2 -11013.138} C_VEL
LIN {X 0,Y 402.818,Z 810.739,A -85,B 0,C 180,E1 -11015.152,E2 -11015.152} C_VEL
LIN {X 0,Y 402.848,Z 810.125,A -85,B 0,C 180,E1 -11016.632,E2 -11016.632} C_VEL
LIN {X 0,Y 402.942,Z 808.355,A -85,B 0,C 180,E1 -11018.293,E2 -11018.293} C_VEL
LIN {X 0,Y 403.228,Z 804.972,A -85,B 0,C 180,E1 -11020.157,E2 -11020.157} C_VEL
LIN {X 0,Y 403.506,Z 799.735,A -85,B 0,C 180,E1 -11022.11,E2 -11022.11} C_VEL
LIN {X 0,Y 403.923,Z 793.567,A -85,B 0,C 180,E1 -11023.802,E2 -11023.802} C_VEL
LIN {X 0,Y 404.485,Z 785.989,A -85,B 0,C 180,E1 -11025.429,E2 -11025.429} C_VEL
LIN {X 0,Y 405.106,Z 778.151,A -85,B 0,C 180,E1 -11026.772,E2 -11026.772} C_VEL
LIN {X 0,Y 405.822,Z 768.407,A -85,B 0,C 180,E1 -11028.131,E2 -11028.131} C_VEL
LIN {X 0,Y 406.558,Z 757.682,A -85,B 0,C 180,E1 -11029.333,E2 -11029.333} C_VEL
LIN {X 0,Y 407.304,Z 746.456,A -85,B 0,C 180,E1 -11030.327,E2 -11030.327} C_VEL
LIN {X 0,Y 407.923,Z 735.16,A -85,B 0,C 180,E1 -11031.116,E2 -11031.116} C_VEL
LIN {X 0,Y 408.459,Z 722.152,A -85,B 0,C 180,E1 -11031.799,E2 -11031.799} C_VEL
LIN {X 0,Y 408.803,Z 709.207,A -85,B 0,C 180,E1 -11032.262,E2 -11032.262} C_VEL
LIN {X 0,Y 409.235,Z 684.254,A -85,B 0,C 180,E1 -11032.769,E2 -11032.769} C_VEL
LIN {X 0,Y 410.157,Z 619.371,A -85,B 0,C 180,E1 -11033.994,E2 -11033.994} C_VEL
LIN {X 0,Y 407.085,Z 606.375,A -85,B 0,C 180,E1 -11034.392,E2 -11034.392} C_VEL
LIN {X 0,Y 405.209,Z 600.49,A -85,B 0,C 180,E1 -11034.605,E2 -11034.605} C_VEL
LIN {X 0,Y 404.186,Z 595.139,A -85,B 0,C 180,E1 -11036.118,E2 -11036.118} C_VEL
LIN {X 0,Y 404.141,Z 595.143,A -85,B 0,C 180,E1 -11039.716,E2 -11039.716} C_VEL
LIN {X 0,Y 404.192,Z 595.133,A -85,B 0,C 180,E1 -11043.124,E2 -11043.124} C_VEL
LIN {X 0,Y 404.174,Z 595.135,A -85,B 0,C 180,E1 -11045.336,E2 -11045.336} C_VEL
LIN {X 0,Y 404.161,Z 595.139,A -85,B 0,C 180,E1 -11048.583,E2 -11048.583} C_VEL
LIN {X 0,Y 404.202,Z 595.132,A -85,B 0,C 180,E1 -11051.932,E2 -11051.932} C_VEL
LIN {X 0,Y 403.507,Z 595.221,A -85,B 0,C 180,E1 -11052.764,E2 -11052.764} C_VEL
LIN {X 0,Y 400.639,Z 595.581,A -85,B 0,C 180,E1 -11054.116,E2 -11054.116} C_VEL
LIN {X 0,Y 398.251,Z 595.875,A -85,B 0,C 180,E1 -11055.209,E2 -11055.209} C_VEL
LIN {X 0,Y 397.26,Z 596.001,A -85,B 0,C 180,E1 -11056.053,E2 -11056.053} C_VEL
LIN {X 0,Y 397.196,Z 596.005,A -85,B 0,C 180,E1 -11056.339,E2 -11056.339} C_VEL
LIN {X 0,Y 397.228,Z 596.002,A -85,B 0,C 180,E1 -11059.81,E2 -11059.81} C_VEL
LIN {X 0,Y 397.364,Z 595.985,A -85,B 0,C 180,E1 -11062.889,E2 -11062.889} C_VEL
LIN {X 0,Y 397.256,Z 595.999,A -85,B 0,C 180,E1 -11064.926,E2 -11064.926} C_VEL
LIN {X 0,Y 397.453,Z 595.974,A -85,B 0,C 180,E1 -11067.974,E2 -11067.974} C_VEL
LIN {X 0,Y 397.58,Z 595.958,A -85,B 0,C 180,E1 -11070.001,E2 -11070.001} C_VEL
LIN {X 0,Y 397.383,Z 595.983,A -85,B 0,C 180,E1 -11073.042,E2 -11073.042} C_VEL
LIN {X 0,Y 397.366,Z 595.985,A -85,B 0,C 180,E1 -11077.113,E2 -11077.113} C_VEL
LIN {X 0,Y 397.221,Z 596.003,A -85,B 0,C 180,E1 -11080.192,E2 -11080.192} C_VEL
LIN {X 0,Y 397.229,Z 596.002,A -85,B 0,C 180,E1 -11083.322,E2 -11083.322} C_VEL
LIN {X 0,Y 397.185,Z 596.009,A -85,B 0,C 180,E1 -11087.156,E2 -11087.156} C_VEL
LIN {X 0,Y 397.106,Z 596.02,A -85,B 0,C 180,E1 -11090.731,E2 -11090.731} C_VEL
LIN {X 0,Y 397.136,Z 596.012,A -85,B 0,C 180,E1 -11094.019,E2 -11094.019} C_VEL
LIN {X 0,Y 397.198,Z 596.007,A -85,B 0,C 180,E1 -11097.391,E2 -11097.391} C_VEL
LIN {X 0,Y 397.083,Z 596.023,A -85,B 0,C 180,E1 -11100.883,E2 -11100.883} C_VEL
LIN {X 0,Y 397.129,Z 596.013,A -85,B 0,C 180,E1 -11104.494,E2 -11104.494} C_VEL
LIN {X 0,Y 397.107,Z 596.015,A -85,B 0,C 180,E1 -11108.276,E2 -11108.276} C_VEL
LIN {X 0,Y 397.093,Z 596.02,A -85,B 0,C 180,E1 -11110.909,E2 -11110.909} C_VEL
LIN {X 0,Y 397.105,Z 596.019,A -85,B 0,C 180,E1 -11113.649,E2 -11113.649} C_VEL
LIN {X 0,Y 397.106,Z 596.015,A -85,B 0,C 180,E1 -11116.522,E2 -11116.522} C_VEL
LIN {X 0,Y 397.117,Z 596.014,A -85,B 0,C 180,E1 -11120.423,E2 -11120.423} C_VEL
LIN {X 0,Y 397.112,Z 596.015,A -85,B 0,C 180,E1 -11124.266,E2 -11124.266} C_VEL
LIN {X 0,Y 397.119,Z 596.014,A -85,B 0,C 180,E1 -11126.728,E2 -11126.728} C_VEL
LIN {X 0,Y 397.129,Z 596.013,A -85,B 0,C 180,E1 -11130.296,E2 -11130.296} C_VEL
LIN {X 0,Y 397.199,Z 596.004,A -85,B 0,C 180,E1 -11132.61,E2 -11132.61} C_VEL
LIN {X 0,Y 397.133,Z 596.016,A -85,B 0,C 180,E1 -11135.982,E2 -11135.982} C_VEL
LIN {X 0,Y 397.144,Z 596.017,A -85,B 0,C 180,E1 -11139.705,E2 -11139.705} C_VEL
LIN {X 0,Y 397.187,Z 596.005,A -85,B 0,C 180,E1 -11142.845,E2 -11142.845} C_VEL
LIN {X 0,Y 397.234,Z 596,A -85,B 0,C 180,E1 -11146.703,E2 -11146.703} C_VEL
LIN {X 0,Y 397.222,Z 596.006,A -85,B 0,C 180,E1 -11149.809,E2 -11149.809} C_VEL
LIN {X 0,Y 397.356,Z 595.984,A -85,B 0,C 180,E1 -11152.888,E2 -11152.888} C_VEL
LIN {X 0,Y 397.258,Z 595.997,A -85,B 0,C 180,E1 -11154.925,E2 -11154.925} C_VEL
LIN {X 0,Y 397.455,Z 595.977,A -85,B 0,C 180,E1 -11157.973,E2 -11157.973} C_VEL
LIN {X 0,Y 397.585,Z 595.961,A -85,B 0,C 180,E1 -11160,E2 -11160} C_VEL
LIN {X 0,Y 397.381,Z 595.981,A -85,B 0,C 180,E1 -11163.042,E2 -11163.042} C_VEL
LIN {X 0,Y 397.379,Z 595.986,A -85,B 0,C 180,E1 -11166.092,E2 -11166.092} C_VEL
LIN {X 0,Y 397.258,Z 595.997,A -85,B 0,C 180,E1 -11169.162,E2 -11169.162} C_VEL
LIN {X 0,Y 397.225,Z 596.006,A -85,B 0,C 180,E1 -11172.258,E2 -11172.258} C_VEL
LIN {X 0,Y 397.185,Z 596.005,A -85,B 0,C 180,E1 -11175.392,E2 -11175.392} C_VEL
LIN {X 0,Y 397.164,Z 596.015,A -85,B 0,C 180,E1 -11178.574,E2 -11178.574} C_VEL
LIN {X 0,Y 397.102,Z 596.016,A -85,B 0,C 180,E1 -11181.818,E2 -11181.818} C_VEL
LIN {X 0,Y 397.158,Z 596.009,A -85,B 0,C 180,E1 -11185.512,E2 -11185.512} C_VEL
LIN {X 0,Y 397.128,Z 596.018,A -85,B 0,C 180,E1 -11188.543,E2 -11188.543} C_VEL
LIN {X 0,Y 397.084,Z 596.019,A -85,B 0,C 180,E1 -11192.071,E2 -11192.071} C_VEL
LIN {X 0,Y 397.125,Z 596.014,A -85,B 0,C 180,E1 -11195.503,E2 -11195.503} C_VEL
LIN {X 0,Y 397.134,Z 596.019,A -85,B 0,C 180,E1 -11198.861,E2 -11198.861} C_VEL
LIN {X 0,Y 397.074,Z 596.02,A -85,B 0,C 180,E1 -11202.267,E2 -11202.267} C_VEL
LIN {X 0,Y 397.093,Z 596.024,A -85,B 0,C 180,E1 -11205.068,E2 -11205.068} C_VEL
LIN {X 0,Y 397.071,Z 596.02,A -85,B 0,C 180,E1 -11208.021,E2 -11208.021} C_VEL
LIN {X 0,Y 397.135,Z 596.019,A -85,B 0,C 180,E1 -11211.138,E2 -11211.138} C_VEL
LIN {X 0,Y 397.125,Z 596.014,A -85,B 0,C 180,E1 -11214.496,E2 -11214.496} C_VEL
LIN {X 0,Y 397.083,Z 596.022,A -85,B 0,C 180,E1 -11217.928,E2 -11217.928} C_VEL
LIN {X 0,Y 397.119,Z 596.059,A -85,B 0,C 180,E1 -11220.228,E2 -11220.228} C_VEL
LIN {X 0,Y 400.18,Z 610.03,A -85,B 0,C 180,E1 -11223.298,E2 -11223.298} C_VEL
LIN {X 0,Y 400.984,Z 616.099,A -85,B 0,C 180,E1 -11224.569,E2 -11224.569} C_VEL
LIN {X 0,Y 399.583,Z 633.901,A -85,B 0,C 180,E1 -11228.052,E2 -11228.052} C_VEL
LIN {X 0,Y 398.875,Z 644.721,A -85,B 0,C 180,E1 -11230.105,E2 -11230.105} C_VEL
LIN {X 0,Y 403.029,Z 674.534,A -85,B 0,C 180,E1 -11230.895,E2 -11230.895} C_VEL
LIN {X 0,Y 401.777,Z 753.506,A -85,B 0,C 180,E1 -11232.437,E2 -11232.437} C_VEL
LIN {X 0,Y 401.235,Z 767.152,A -85,B 0,C 180,E1 -11232.905,E2 -11232.905} C_VEL
LIN {X 0,Y 400.514,Z 780.092,A -85,B 0,C 180,E1 -11233.562,E2 -11233.562} C_VEL
LIN {X 0,Y 399.645,Z 792.7,A -85,B 0,C 180,E1 -11234.443,E2 -11234.443} C_VEL
LIN {X 0,Y 398.889,Z 803.993,A -85,B 0,C 180,E1 -11235.458,E2 -11235.458} C_VEL
LIN {X 0,Y 398.074,Z 815.146,A -85,B 0,C 180,E1 -11236.73,E2 -11236.73} C_VEL
LIN {X 0,Y 397.389,Z 824.171,A -85,B 0,C 180,E1 -11238.005,E2 -11238.005} C_VEL
LIN {X 0,Y 396.677,Z 832.968,A -85,B 0,C 180,E1 -11239.536,E2 -11239.536} C_VEL
LIN {X 0,Y 396.31,Z 839.986,A -85,B 0,C 180,E1 -11241.072,E2 -11241.072} C_VEL
LIN {X 0,Y 396.004,Z 846.416,A -85,B 0,C 180,E1 -11242.863,E2 -11242.863} C_VEL
LIN {X 0,Y 395.87,Z 850.606,A -85,B 0,C 180,E1 -11244.395,E2 -11244.395} C_VEL
LIN {X 0,Y 395.813,Z 853.701,A -85,B 0,C 180,E1 -11245.926,E2 -11245.926} C_VEL
LIN {X 0,Y 395.854,Z 855.223,A -85,B 0,C 180,E1 -11246.946,E2 -11246.946} C_VEL
LIN {X 0,Y 395.916,Z 856.277,A -85,B 0,C 180,E1 -11247.964,E2 -11247.964} C_VEL
LIN {X 0,Y 395.874,Z 856.917,A -85,B 0,C 180,E1 -11248.982,E2 -11248.982} C_VEL
LIN {X 0,Y 395.874,Z 857.159,A -85,B 0,C 180,E1 -11249.999,E2 -11249.999} C_VEL
LIN {X 0,Y 395.874,Z 856.979,A -85,B 0,C 180,E1 -11251.016,E2 -11251.016} C_VEL
LIN {X 0,Y 395.917,Z 856.357,A -85,B 0,C 180,E1 -11252.033,E2 -11252.033} C_VEL
LIN {X 0,Y 395.852,Z 855.326,A -85,B 0,C 180,E1 -11253.052,E2 -11253.052} C_VEL
LIN {X 0,Y 395.809,Z 853.89,A -85,B 0,C 180,E1 -11254.072,E2 -11254.072} C_VEL
LIN {X 0,Y 395.841,Z 850.364,A -85,B 0,C 180,E1 -11255.824,E2 -11255.824} C_VEL
LIN {X 0,Y 396.057,Z 845.183,A -85,B 0,C 180,E1 -11257.647,E2 -11257.647} C_VEL
LIN {X 0,Y 396.439,Z 838.477,A -85,B 0,C 180,E1 -11259.437,E2 -11259.437} C_VEL
LIN {X 0,Y 396.91,Z 831.13,A -85,B 0,C 180,E1 -11260.972,E2 -11260.972} C_VEL
LIN {X 0,Y 397.703,Z 822.017,A -85,B 0,C 180,E1 -11262.501,E2 -11262.501} C_VEL
LIN {X 0,Y 398.435,Z 812.681,A -85,B 0,C 180,E1 -11263.775,E2 -11263.775} C_VEL
LIN {X 0,Y 399.243,Z 802.342,A -85,B 0,C 180,E1 -11264.917,E2 -11264.917} C_VEL
LIN {X 0,Y 400.117,Z 790.913,A -85,B 0,C 180,E1 -11265.928,E2 -11265.928} C_VEL
LIN {X 0,Y 400.994,Z 779.134,A -85,B 0,C 180,E1 -11266.742,E2 -11266.742} C_VEL
LIN {X 0,Y 401.78,Z 767.167,A -85,B 0,C 180,E1 -11267.364,E2 -11267.364} C_VEL
LIN {X 0,Y 402.389,Z 754.289,A -85,B 0,C 180,E1 -11267.829,E2 -11267.829} C_VEL
LIN {X 0,Y 402.891,Z 731.086,A -85,B 0,C 180,E1 -11268.321,E2 -11268.321} C_VEL
LIN {X 0,Y 403.729,Z 674.205,A -85,B 0,C 180,E1 -11269.454,E2 -11269.454} C_VEL
LIN {X 0,Y 400.411,Z 650.01,A -85,B 0,C 180,E1 -11270.155,E2 -11270.155} C_VEL
LIN {X 0,Y 399.086,Z 642.45,A -85,B 0,C 180,E1 -11270.399,E2 -11270.399} C_VEL
LIN {X 0,Y 400.625,Z 623.324,A -85,B 0,C 180,E1 -11274.186,E2 -11274.186} C_VEL
LIN {X 0,Y 401.219,Z 615.874,A -85,B 0,C 180,E1 -11275.691,E2 -11275.691} C_VEL
LIN {X 0,Y 399.591,Z 606.601,A -85,B 0,C 180,E1 -11277.773,E2 -11277.773} C_VEL
LIN {X 0,Y 397.122,Z 596.025,A -85,B 0,C 180,E1 -11280.331,E2 -11280.331} C_VEL
LIN {X 0,Y 397.116,Z 596.02,A -85,B 0,C 180,E1 -11283.717,E2 -11283.717} C_VEL
LIN {X 0,Y 397.095,Z 596.021,A -85,B 0,C 180,E1 -11287.209,E2 -11287.209} C_VEL
LIN {X 0,Y 397.116,Z 596.023,A -85,B 0,C 180,E1 -11290.448,E2 -11290.448} C_VEL
LIN {X 0,Y 397.099,Z 596.022,A -85,B 0,C 180,E1 -11293.647,E2 -11293.647} C_VEL
LIN {X 0,Y 397.159,Z 596.014,A -85,B 0,C 180,E1 -11296.51,E2 -11296.51} C_VEL
LIN {X 0,Y 397.118,Z 596.016,A -85,B 0,C 180,E1 -11299.55,E2 -11299.55} C_VEL
LIN {X 0,Y 397.093,Z 596.019,A -85,B 0,C 180,E1 -11302.789,E2 -11302.789} C_VEL
LIN {X 0,Y 397.112,Z 596.017,A -85,B 0,C 180,E1 -11306.281,E2 -11306.281} C_VEL
LIN {X 0,Y 397.085,Z 596.018,A -85,B 0,C 180,E1 -11309.118,E2 -11309.118} C_VEL
LIN {X 0,Y 397.187,Z 596.009,A -85,B 0,C 180,E1 -11312.609,E2 -11312.609} C_VEL
LIN {X 0,Y 397.125,Z 596.016,A -85,B 0,C 180,E1 -11315.981,E2 -11315.981} C_VEL
LIN {X 0,Y 397.13,Z 596.012,A -85,B 0,C 180,E1 -11319.704,E2 -11319.704} C_VEL
LIN {X 0,Y 397.173,Z 596.011,A -85,B 0,C 180,E1 -11322.844,E2 -11322.844} C_VEL
LIN {X 0,Y 397.218,Z 596.006,A -85,B 0,C 180,E1 -11326.678,E2 -11326.678} C_VEL
LIN {X 0,Y 397.22,Z 596.005,A -85,B 0,C 180,E1 -11329.809,E2 -11329.809} C_VEL
LIN {X 0,Y 397.355,Z 595.988,A -85,B 0,C 180,E1 -11332.888,E2 -11332.888} C_VEL
LIN {X 0,Y 397.248,Z 596.001,A -85,B 0,C 180,E1 -11334.925,E2 -11334.925} C_VEL
LIN {X 0,Y 397.443,Z 595.979,A -85,B 0,C 180,E1 -11337.973,E2 -11337.973} C_VEL
LIN {X 0,Y 397.574,Z 595.964,A -85,B 0,C 180,E1 -11340,E2 -11340} C_VEL
LIN {X 0,Y 397.375,Z 595.986,A -85,B 0,C 180,E1 -11343.041,E2 -11343.041} C_VEL
LIN {X 0,Y 397.353,Z 595.99,A -85,B 0,C 180,E1 -11346.603,E2 -11346.603} C_VEL
LIN {X 0,Y 397.25,Z 596.003,A -85,B 0,C 180,E1 -11349.162,E2 -11349.162} C_VEL
LIN {X 0,Y 397.236,Z 596.089,A -85,B 0,C 180,E1 -11352.51,E2 -11352.51} C_VEL
LIN {X 0,Y 398.626,Z 603.171,A -85,B 0,C 180,E1 -11354.648,E2 -11354.648} C_VEL
LIN {X 0,Y 402.679,Z 613.974,A -85,B 0,C 180,E1 -11355.141,E2 -11355.141} C_VEL
LIN {X 0,Y 404.559,Z 622.265,A -85,B 0,C 180,E1 -11355.429,E2 -11355.429} C_VEL
LIN {X 0,Y 402.832,Z 709.492,A -85,B 0,C 180,E1 -11357.181,E2 -11357.181} C_VEL
LIN {X 0,Y 402.429,Z 722.995,A -85,B 0,C 180,E1 -11357.664,E2 -11357.664} C_VEL
LIN {X 0,Y 401.855,Z 734.951,A -85,B 0,C 180,E1 -11358.283,E2 -11358.283} C_VEL
LIN {X 0,Y 401.184,Z 746.799,A -85,B 0,C 180,E1 -11359.111,E2 -11359.111} C_VEL
LIN {X 0,Y 400.383,Z 758.354,A -85,B 0,C 180,E1 -11360.15,E2 -11360.15} C_VEL
LIN {X 0,Y 399.542,Z 767.878,A -85,B 0,C 180,E1 -11361.211,E2 -11361.211} C_VEL
LIN {X 0,Y 398.708,Z 777.539,A -85,B 0,C 180,E1 -11362.543,E2 -11362.543} C_VEL
LIN {X 0,Y 397.916,Z 785.886,A -85,B 0,C 180,E1 -11363.968,E2 -11363.968} C_VEL
LIN {X 0,Y 397.288,Z 793.362,A -85,B 0,C 180,E1 -11365.556,E2 -11365.556} C_VEL
LIN {X 0,Y 396.878,Z 798.224,A -85,B 0,C 180,E1 -11366.844,E2 -11366.844} C_VEL
LIN {X 0,Y 396.432,Z 803.483,A -85,B 0,C 180,E1 -11368.598,E2 -11368.598} C_VEL
LIN {X 0,Y 396.15,Z 807.289,A -85,B 0,C 180,E1 -11370.372,E2 -11370.372} C_VEL
LIN {X 0,Y 395.895,Z 809.817,A -85,B 0,C 180,E1 -11372.179,E2 -11372.179} C_VEL
LIN {X 0,Y 395.758,Z 810.811,A -85,B 0,C 180,E1 -11373.424,E2 -11373.424} C_VEL
LIN {X 0,Y 395.741,Z 811.136,A -85,B 0,C 180,E1 -11375.225,E2 -11375.225} C_VEL
LIN {X 0,Y 395.782,Z 810.117,A -85,B 0,C 180,E1 -11377.139,E2 -11377.139} C_VEL
LIN {X 0,Y 395.892,Z 808.292,A -85,B 0,C 180,E1 -11378.641,E2 -11378.641} C_VEL
LIN {X 0,Y 396.182,Z 805.216,A -85,B 0,C 180,E1 -11380.291,E2 -11380.291} C_VEL
LIN {X 0,Y 396.386,Z 801.146,A -85,B 0,C 180,E1 -11381.871,E2 -11381.871} C_VEL
LIN {X 0,Y 396.726,Z 795.945,A -85,B 0,C 180,E1 -11383.424,E2 -11383.424} C_VEL
LIN {X 0,Y 397.334,Z 789.054,A -85,B 0,C 180,E1 -11385.033,E2 -11385.033} C_VEL
LIN {X 0,Y 397.811,Z 781.537,A -85,B 0,C 180,E1 -11386.451,E2 -11386.451} C_VEL
LIN {X 0,Y 398.561,Z 772.857,A -85,B 0,C 180,E1 -11387.783,E2 -11387.783} C_VEL
LIN {X 0,Y 399.332,Z 763.155,A -85,B 0,C 180,E1 -11388.998,E2 -11388.998} C_VEL
LIN {X 0,Y 400.083,Z 752.333,A -85,B 0,C 180,E1 -11390.086,E2 -11390.086} C_VEL
LIN {X 0,Y 400.811,Z 740.126,A -85,B 0,C 180,E1 -11391.055,E2 -11391.055} C_VEL
LIN {X 0,Y 401.44,Z 727.567,A -85,B 0,C 180,E1 -11391.807,E2 -11391.807} C_VEL
LIN {X 0,Y 401.853,Z 713.988,A -85,B 0,C 180,E1 -11392.383,E2 -11392.383} C_VEL
LIN {X 0,Y 402.213,Z 700.996,A -85,B 0,C 180,E1 -11392.723,E2 -11392.723} C_VEL
LIN {X 0,Y 403.407,Z 620.555,A -85,B 0,C 180,E1 -11394.276,E2 -11394.276} C_VEL
LIN {X 0,Y 400.522,Z 608.377,A -85,B 0,C 180,E1 -11394.656,E2 -11394.656} C_VEL
LIN {X 0,Y 398.055,Z 600.814,A -85,B 0,C 180,E1 -11394.946,E2 -11394.946} C_VEL
LIN {X 0,Y 397.159,Z 596.014,A -85,B 0,C 180,E1 -11396.273,E2 -11396.273} C_VEL
LIN {X 0,Y 397.121,Z 596.017,A -85,B 0,C 180,E1 -11400.297,E2 -11400.297} C_VEL
LIN {X 0,Y 397.191,Z 596.006,A -85,B 0,C 180,E1 -11402.611,E2 -11402.611} C_VEL
LIN {X 0,Y 397.13,Z 596.018,A -85,B 0,C 180,E1 -11405.983,E2 -11405.983} C_VEL
LIN {X 0,Y 397.152,Z 596.012,A -85,B 0,C 180,E1 -11409.7,E2 -11409.7} C_VEL
LIN {X 0,Y 397.18,Z 596.007,A -85,B 0,C 180,E1 -11412.846,E2 -11412.846} C_VEL
LIN {X 0,Y 397.196,Z 596.005,A -85,B 0,C 180,E1 -11416.339,E2 -11416.339} C_VEL
LIN {X 0,Y 396.569,Z 596.087,A -85,B 0,C 180,E1 -11417.185,E2 -11417.185} C_VEL
LIN {X 0,Y 393.719,Z 596.447,A -85,B 0,C 180,E1 -11418.56,E2 -11418.56} C_VEL
LIN {X 0,Y 391.299,Z 596.748,A -85,B 0,C 180,E1 -11419.671,E2 -11419.671} C_VEL
LIN {X 0,Y 390.285,Z 596.87,A -85,B 0,C 180,E1 -11420.531,E2 -11420.531} C_VEL
LIN {X 0,Y 390.217,Z 596.876,A -85,B 0,C 180,E1 -11420.822,E2 -11420.822} C_VEL
LIN {X 0,Y 390.319,Z 596.864,A -85,B 0,C 180,E1 -11422.76,E2 -11422.76} C_VEL
LIN {X 0,Y 390.228,Z 596.875,A -85,B 0,C 180,E1 -11424.835,E2 -11424.835} C_VEL
LIN {X 0,Y 390.422,Z 596.849,A -85,B 0,C 180,E1 -11427.938,E2 -11427.938} C_VEL
LIN {X 0,Y 390.549,Z 596.834,A -85,B 0,C 180,E1 -11430.001,E2 -11430.001} C_VEL
LIN {X 0,Y 390.317,Z 596.863,A -85,B 0,C 180,E1 -11433.098,E2 -11433.098} C_VEL
LIN {X 0,Y 390.332,Z 596.861,A -85,B 0,C 180,E1 -11436.203,E2 -11436.203} C_VEL
LIN {X 0,Y 390.317,Z 596.864,A -85,B 0,C 180,E1 -11438.283,E2 -11438.283} C_VEL
LIN {X 0,Y 390.174,Z 596.883,A -85,B 0,C 180,E1 -11442.484,E2 -11442.484} C_VEL
LIN {X 0,Y 390.142,Z 596.883,A -85,B 0,C 180,E1 -11445.678,E2 -11445.678} C_VEL
LIN {X 0,Y 390.109,Z 596.894,A -85,B 0,C 180,E1 -11448.923,E2 -11448.923} C_VEL
LIN {X 0,Y 390.043,Z 596.896,A -85,B 0,C 180,E1 -11452.235,E2 -11452.235} C_VEL
LIN {X 0,Y 390.123,Z 596.886,A -85,B 0,C 180,E1 -11455.744,E2 -11455.744} C_VEL
LIN {X 0,Y 390.063,Z 596.9,A -85,B 0,C 180,E1 -11459.11,E2 -11459.11} C_VEL
LIN {X 0,Y 390.047,Z 596.897,A -85,B 0,C 180,E1 -11462.722,E2 -11462.722} C_VEL
LIN {X 0,Y 390.06,Z 596.894,A -85,B 0,C 180,E1 -11465.826,E2 -11465.826} C_VEL
LIN {X 0,Y 390.075,Z 596.898,A -85,B 0,C 180,E1 -11469.219,E2 -11469.219} C_VEL
LIN {X 0,Y 390.046,Z 596.895,A -85,B 0,C 180,E1 -11472.375,E2 -11472.375} C_VEL
LIN {X 0,Y 390.048,Z 596.902,A -85,B 0,C 180,E1 -11475.355,E2 -11475.355} C_VEL
LIN {X 0,Y 390.035,Z 596.897,A -85,B 0,C 180,E1 -11478.187,E2 -11478.187} C_VEL
LIN {X 0,Y 390.091,Z 596.891,A -85,B 0,C 180,E1 -11480.908,E2 -11480.908} C_VEL
LIN {X 0,Y 390.089,Z 596.89,A -85,B 0,C 180,E1 -11484.794,E2 -11484.794} C_VEL
LIN {X 0,Y 390.028,Z 596.897,A -85,B 0,C 180,E1 -11488.496,E2 -11488.496} C_VEL
LIN {X 0,Y 390.122,Z 596.888,A -85,B 0,C 180,E1 -11492.07,E2 -11492.07} C_VEL
LIN {X 0,Y 390.082,Z 596.895,A -85,B 0,C 180,E1 -11495.52,E2 -11495.52} C_VEL
LIN {X 0,Y 390.093,Z 596.893,A -85,B 0,C 180,E1 -11499.53,E2 -11499.53} C_VEL
LIN {X 0,Y 390.143,Z 596.884,A -85,B 0,C 180,E1 -11503.249,E2 -11503.249} C_VEL
LIN {X 0,Y 390.2,Z 596.877,A -85,B 0,C 180,E1 -11506.562,E2 -11506.562} C_VEL
LIN {X 0,Y 390.21,Z 596.875,A -85,B 0,C 180,E1 -11510.671,E2 -11510.671} C_VEL
LIN {X 0,Y 390.33,Z 596.863,A -85,B 0,C 180,E1 -11513.798,E2 -11513.798} C_VEL
LIN {X 0,Y 390.423,Z 596.852,A -85,B 0,C 180,E1 -11517.937,E2 -11517.937} C_VEL
LIN {X 0,Y 390.554,Z 596.837,A -85,B 0,C 180,E1 -11520,E2 -11520} C_VEL
LIN {X 0,Y 390.315,Z 596.861,A -85,B 0,C 180,E1 -11523.097,E2 -11523.097} C_VEL
LIN {X 0,Y 390.333,Z 596.865,A -85,B 0,C 180,E1 -11526.202,E2 -11526.202} C_VEL
LIN {X 0,Y 390.211,Z 596.874,A -85,B 0,C 180,E1 -11529.329,E2 -11529.329} C_VEL
LIN {X 0,Y 390.201,Z 596.875,A -85,B 0,C 180,E1 -11533.438,E2 -11533.438} C_VEL
LIN {X 0,Y 390.135,Z 596.884,A -85,B 0,C 180,E1 -11537.298,E2 -11537.298} C_VEL
LIN {X 0,Y 390.093,Z 596.895,A -85,B 0,C 180,E1 -11540.47,E2 -11540.47} C_VEL
LIN {X 0,Y 390.084,Z 596.896,A -85,B 0,C 180,E1 -11544.481,E2 -11544.481} C_VEL
LIN {X 0,Y 390.123,Z 596.886,A -85,B 0,C 180,E1 -11547.93,E2 -11547.93} C_VEL
LIN {X 0,Y 390.029,Z 596.897,A -85,B 0,C 180,E1 -11551.504,E2 -11551.504} C_VEL
LIN {X 0,Y 390.091,Z 596.892,A -85,B 0,C 180,E1 -11555.207,E2 -11555.207} C_VEL
LIN {X 0,Y 390.074,Z 596.895,A -85,B 0,C 180,E1 -11559.218,E2 -11559.218} C_VEL
LIN {X 0,Y 390.048,Z 596.896,A -85,B 0,C 180,E1 -11562.374,E2 -11562.374} C_VEL
LIN {X 0,Y 390.05,Z 596.898,A -85,B 0,C 180,E1 -11565.354,E2 -11565.354} C_VEL
LIN {X 0,Y 390.036,Z 596.896,A -85,B 0,C 180,E1 -11568.186,E2 -11568.186} C_VEL
LIN {X 0,Y 390.095,Z 596.893,A -85,B 0,C 180,E1 -11570.907,E2 -11570.907} C_VEL
LIN {X 0,Y 390.09,Z 596.892,A -85,B 0,C 180,E1 -11574.793,E2 -11574.793} C_VEL
LIN {X 0,Y 390.029,Z 596.9,A -85,B 0,C 180,E1 -11578.495,E2 -11578.495} C_VEL
LIN {X 0,Y 390.083,Z 597.017,A -85,B 0,C 180,E1 -11579.966,E2 -11579.966} C_VEL
LIN {X 0,Y 393.217,Z 611.281,A -85,B 0,C 180,E1 -11583.165,E2 -11583.165} C_VEL
LIN {X 0,Y 394.04,Z 616.915,A -85,B 0,C 180,E1 -11584.372,E2 -11584.372} C_VEL
LIN {X 0,Y 392.692,Z 633.354,A -85,B 0,C 180,E1 -11587.646,E2 -11587.646} C_VEL
LIN {X 0,Y 391.904,Z 644.135,A -85,B 0,C 180,E1 -11589.77,E2 -11589.77} C_VEL
LIN {X 0,Y 396.229,Z 675.133,A -85,B 0,C 180,E1 -11590.613,E2 -11590.613} C_VEL
LIN {X 0,Y 394.902,Z 753.75,A -85,B 0,C 180,E1 -11592.188,E2 -11592.188} C_VEL
LIN {X 0,Y 394.352,Z 767.179,A -85,B 0,C 180,E1 -11592.664,E2 -11592.664} C_VEL
LIN {X 0,Y 393.576,Z 779.967,A -85,B 0,C 180,E1 -11593.331,E2 -11593.331} C_VEL
LIN {X 0,Y 392.777,Z 791.728,A -85,B 0,C 180,E1 -11594.164,E2 -11594.164} C_VEL
LIN {X 0,Y 391.96,Z 803.121,A -85,B 0,C 180,E1 -11595.195,E2 -11595.195} C_VEL
LIN {X 0,Y 391.209,Z 813.197,A -85,B 0,C 180,E1 -11596.333,E2 -11596.333} C_VEL
LIN {X 0,Y 390.527,Z 821.833,A -85,B 0,C 180,E1 -11597.527,E2 -11597.527} C_VEL
LIN {X 0,Y 389.77,Z 830.984,A -85,B 0,C 180,E1 -11599.085,E2 -11599.085} C_VEL
LIN {X 0,Y 389.302,Z 838.36,A -85,B 0,C 180,E1 -11600.648,E2 -11600.648} C_VEL
LIN {X 0,Y 388.993,Z 844.239,A -85,B 0,C 180,E1 -11602.211,E2 -11602.211} C_VEL
LIN {X 0,Y 388.836,Z 848.846,A -85,B 0,C 180,E1 -11603.773,E2 -11603.773} C_VEL
LIN {X 0,Y 388.808,Z 851.263,A -85,B 0,C 180,E1 -11604.814,E2 -11604.814} C_VEL
LIN {X 0,Y 388.737,Z 853.231,A -85,B 0,C 180,E1 -11605.852,E2 -11605.852} C_VEL
LIN {X 0,Y 388.757,Z 854.769,A -85,B 0,C 180,E1 -11606.89,E2 -11606.89} C_VEL
LIN {X 0,Y 388.846,Z 855.839,A -85,B 0,C 180,E1 -11607.927,E2 -11607.927} C_VEL
LIN {X 0,Y 388.802,Z 856.488,A -85,B 0,C 180,E1 -11608.963,E2 -11608.963} C_VEL
LIN {X 0,Y 388.798,Z 856.738,A -85,B 0,C 180,E1 -11609.999,E2 -11609.999} C_VEL
LIN {X 0,Y 388.802,Z 856.574,A -85,B 0,C 180,E1 -11611.035,E2 -11611.035} C_VEL
LIN {X 0,Y 388.847,Z 855.962,A -85,B 0,C 180,E1 -11612.07,E2 -11612.07} C_VEL
LIN {X 0,Y 388.753,Z 854.938,A -85,B 0,C 180,E1 -11613.108,E2 -11613.108} C_VEL
LIN {X 0,Y 388.732,Z 853.508,A -85,B 0,C 180,E1 -11614.146,E2 -11614.146} C_VEL
LIN {X 0,Y 388.743,Z 850.355,A -85,B 0,C 180,E1 -11615.775,E2 -11615.775} C_VEL
LIN {X 0,Y 388.93,Z 846.449,A -85,B 0,C 180,E1 -11617.266,E2 -11617.266} C_VEL
LIN {X 0,Y 389.237,Z 840.229,A -85,B 0,C 180,E1 -11619.089,E2 -11619.089} C_VEL
LIN {X 0,Y 389.678,Z 833.415,A -85,B 0,C 180,E1 -11620.652,E2 -11620.652} C_VEL
LIN {X 0,Y 390.436,Z 824.979,A -85,B 0,C 180,E1 -11622.209,E2 -11622.209} C_VEL
LIN {X 0,Y 391.279,Z 815.137,A -85,B 0,C 180,E1 -11623.67,E2 -11623.67} C_VEL
LIN {X 0,Y 392.146,Z 804.613,A -85,B 0,C 180,E1 -11624.928,E2 -11624.928} C_VEL
LIN {X 0,Y 393.051,Z 793.944,A -85,B 0,C 180,E1 -11625.956,E2 -11625.956} C_VEL
LIN {X 0,Y 394.04,Z 782.147,A -85,B 0,C 180,E1 -11626.847,E2 -11626.847} C_VEL
LIN {X 0,Y 394.73,Z 771.294,A -85,B 0,C 180,E1 -11627.483,E2 -11627.483} C_VEL
LIN {X 0,Y 395.526,Z 757.873,A -85,B 0,C 180,E1 -11628.048,E2 -11628.048} C_VEL
LIN {X 0,Y 395.912,Z 744.859,A -85,B 0,C 180,E1 -11628.398,E2 -11628.398} C_VEL
LIN {X 0,Y 397.108,Z 674.866,A -85,B 0,C 180,E1 -11629.812,E2 -11629.812} C_VEL
LIN {X 0,Y 393.876,Z 651.149,A -85,B 0,C 180,E1 -11630.524,E2 -11630.524} C_VEL
LIN {X 0,Y 392.266,Z 641.794,A -85,B 0,C 180,E1 -11630.864,E2 -11630.864} C_VEL
LIN {X 0,Y 393.782,Z 623.99,A -85,B 0,C 180,E1 -11634.464,E2 -11634.464} C_VEL
LIN {X 0,Y 394.343,Z 617.115,A -85,B 0,C 180,E1 -11635.888,E2 -11635.888} C_VEL
LIN {X 0,Y 392.572,Z 607.355,A -85,B 0,C 180,E1 -11638.138,E2 -11638.138} C_VEL
LIN {X 0,Y 390.058,Z 596.904,A -85,B 0,C 180,E1 -11640.746,E2 -11640.746} C_VEL
LIN {X 0,Y 390.065,Z 596.898,A -85,B 0,C 180,E1 -11644.023,E2 -11644.023} C_VEL
LIN {X 0,Y 390.044,Z 596.899,A -85,B 0,C 180,E1 -11647.55,E2 -11647.55} C_VEL
LIN {X 0,Y 390.073,Z 596.899,A -85,B 0,C 180,E1 -11650.824,E2 -11650.824} C_VEL
LIN {X 0,Y 390.055,Z 596.901,A -85,B 0,C 180,E1 -11653.886,E2 -11653.886} C_VEL
LIN {X 0,Y 390.112,Z 596.892,A -85,B 0,C 180,E1 -11656.797,E2 -11656.797} C_VEL
LIN {X 0,Y 390.073,Z 596.894,A -85,B 0,C 180,E1 -11659.562,E2 -11659.562} C_VEL
LIN {X 0,Y 390.041,Z 596.902,A -85,B 0,C 180,E1 -11662.447,E2 -11662.447} C_VEL
LIN {X 0,Y 390.077,Z 596.892,A -85,B 0,C 180,E1 -11666.046,E2 -11666.046} C_VEL
LIN {X 0,Y 390.046,Z 596.895,A -85,B 0,C 180,E1 -11669.701,E2 -11669.701} C_VEL
LIN {X 0,Y 390.106,Z 596.886,A -85,B 0,C 180,E1 -11673.231,E2 -11673.231} C_VEL
LIN {X 0,Y 390.099,Z 596.889,A -85,B 0,C 180,E1 -11676.75,E2 -11676.75} C_VEL
LIN {X 0,Y 390.096,Z 596.889,A -85,B 0,C 180,E1 -11679.982,E2 -11679.982} C_VEL
LIN {X 0,Y 390.13,Z 596.887,A -85,B 0,C 180,E1 -11683.248,E2 -11683.248} C_VEL
LIN {X 0,Y 390.186,Z 596.883,A -85,B 0,C 180,E1 -11686.561,E2 -11686.561} C_VEL
LIN {X 0,Y 390.17,Z 596.883,A -85,B 0,C 180,E1 -11689.623,E2 -11689.623} C_VEL
LIN {X 0,Y 390.31,Z 596.866,A -85,B 0,C 180,E1 -11692.759,E2 -11692.759} C_VEL
LIN {X 0,Y 390.22,Z 596.876,A -85,B 0,C 180,E1 -11694.833,E2 -11694.833} C_VEL
LIN {X 0,Y 390.412,Z 596.855,A -85,B 0,C 180,E1 -11697.937,E2 -11697.937} C_VEL
LIN {X 0,Y 390.543,Z 596.839,A -85,B 0,C 180,E1 -11700,E2 -11700} C_VEL
LIN {X 0,Y 390.309,Z 596.866,A -85,B 0,C 180,E1 -11703.096,E2 -11703.096} C_VEL
LIN {X 0,Y 390.309,Z 596.868,A -85,B 0,C 180,E1 -11706.598,E2 -11706.598} C_VEL
LIN {X 0,Y 390.306,Z 596.87,A -85,B 0,C 180,E1 -11708.282,E2 -11708.282} C_VEL
LIN {X 0,Y 390.218,Z 597.076,A -85,B 0,C 180,E1 -11712.151,E2 -11712.151} C_VEL
LIN {X 0,Y 391.553,Z 603.76,A -85,B 0,C 180,E1 -11714.207,E2 -11714.207} C_VEL
LIN {X 0,Y 396.335,Z 616.111,A -85,B 0,C 180,E1 -11714.794,E2 -11714.794} C_VEL
LIN {X 0,Y 398.012,Z 623.34,A -85,B 0,C 180,E1 -11715.059,E2 -11715.059} C_VEL
LIN {X 0,Y 396.175,Z 710.186,A -85,B 0,C 180,E1 -11716.845,E2 -11716.845} C_VEL
LIN {X 0,Y 395.748,Z 723.511,A -85,B 0,C 180,E1 -11717.332,E2 -11717.332} C_VEL
LIN {X 0,Y 395.104,Z 736.116,A -85,B 0,C 180,E1 -11718.003,E2 -11718.003} C_VEL
LIN {X 0,Y 394.414,Z 747.553,A -85,B 0,C 180,E1 -11718.825,E2 -11718.825} C_VEL
LIN {X 0,Y 393.614,Z 758.558,A -85,B 0,C 180,E1 -11719.831,E2 -11719.831} C_VEL
LIN {X 0,Y 392.678,Z 768.66,A -85,B 0,C 180,E1 -11720.974,E2 -11720.974} C_VEL
LIN {X 0,Y 391.743,Z 778.734,A -85,B 0,C 180,E1 -11722.41,E2 -11722.41} C_VEL
LIN {X 0,Y 390.879,Z 787.451,A -85,B 0,C 180,E1 -11723.958,E2 -11723.958} C_VEL
LIN {X 0,Y 390.243,Z 794.78,A -85,B 0,C 180,E1 -11725.609,E2 -11725.609} C_VEL
LIN {X 0,Y 389.679,Z 800.777,A -85,B 0,C 180,E1 -11727.332,E2 -11727.332} C_VEL
LIN {X 0,Y 389.248,Z 805.616,A -85,B 0,C 180,E1 -11729.176,E2 -11729.176} C_VEL
LIN {X 0,Y 389.075,Z 807.928,A -85,B 0,C 180,E1 -11730.383,E2 -11730.383} C_VEL
LIN {X 0,Y 388.855,Z 809.983,A -85,B 0,C 180,E1 -11731.85,E2 -11731.85} C_VEL
LIN {X 0,Y 388.649,Z 811.384,A -85,B 0,C 180,E1 -11733.716,E2 -11733.716} C_VEL
LIN {X 0,Y 388.654,Z 811.486,A -85,B 0,C 180,E1 -11735.54,E2 -11735.54} C_VEL
LIN {X 0,Y 388.718,Z 810.4,A -85,B 0,C 180,E1 -11737.298,E2 -11737.298} C_VEL
LIN {X 0,Y 388.897,Z 807.794,A -85,B 0,C 180,E1 -11739.235,E2 -11739.235} C_VEL
LIN {X 0,Y 389.13,Z 804.921,A -85,B 0,C 180,E1 -11740.665,E2 -11740.665} C_VEL
LIN {X 0,Y 389.371,Z 800.616,A -85,B 0,C 180,E1 -11742.268,E2 -11742.268} C_VEL
LIN {X 0,Y 389.797,Z 795.126,A -85,B 0,C 180,E1 -11743.849,E2 -11743.849} C_VEL
LIN {X 0,Y 390.347,Z 788.359,A -85,B 0,C 180,E1 -11745.4,E2 -11745.4} C_VEL
LIN {X 0,Y 391.045,Z 780.09,A -85,B 0,C 180,E1 -11746.927,E2 -11746.927} C_VEL
LIN {X 0,Y 391.671,Z 772.117,A -85,B 0,C 180,E1 -11748.13,E2 -11748.13} C_VEL
LIN {X 0,Y 392.468,Z 762.14,A -85,B 0,C 180,E1 -11749.36,E2 -11749.36} C_VEL
LIN {X 0,Y 393.227,Z 751.485,A -85,B 0,C 180,E1 -11750.422,E2 -11750.422} C_VEL
LIN {X 0,Y 393.991,Z 739.485,A -85,B 0,C 180,E1 -11751.369,E2 -11751.369} C_VEL
LIN {X 0,Y 394.586,Z 727.415,A -85,B 0,C 180,E1 -11752.087,E2 -11752.087} C_VEL
LIN {X 0,Y 395.039,Z 713.683,A -85,B 0,C 180,E1 -11752.671,E2 -11752.671} C_VEL
LIN {X 0,Y 395.405,Z 699.264,A -85,B 0,C 180,E1 -11753.034,E2 -11753.034} C_VEL
LIN {X 0,Y 396.61,Z 621.496,A -85,B 0,C 180,E1 -11754.566,E2 -11754.566} C_VEL
LIN {X 0,Y 393.976,Z 610.444,A -85,B 0,C 180,E1 -11754.92,E2 -11754.92} C_VEL
LIN {X 0,Y 390.942,Z 601.274,A -85,B 0,C 180,E1 -11755.265,E2 -11755.265} C_VEL
LIN {X 0,Y 390.115,Z 596.89,A -85,B 0,C 180,E1 -11756.517,E2 -11756.517} C_VEL
LIN {X 0,Y 390.043,Z 596.901,A -85,B 0,C 180,E1 -11759.87,E2 -11759.87} C_VEL
LIN {X 0,Y 390.11,Z 596.887,A -85,B 0,C 180,E1 -11763.233,E2 -11763.233} C_VEL
LIN {X 0,Y 390.104,Z 596.889,A -85,B 0,C 180,E1 -11766.751,E2 -11766.751} C_VEL
LIN {X 0,Y 390.118,Z 596.891,A -85,B 0,C 180,E1 -11769.985,E2 -11769.985} C_VEL
LIN {X 0,Y 390.137,Z 596.883,A -85,B 0,C 180,E1 -11773.249,E2 -11773.249} C_VEL
LIN {X 0,Y 390.193,Z 596.881,A -85,B 0,C 180,E1 -11776.563,E2 -11776.563} C_VEL
LIN {X 0,Y 390.178,Z 596.879,A -85,B 0,C 180,E1 -11779.624,E2 -11779.624} C_VEL
LIN {X 0,Y 390.217,Z 596.876,A -85,B 0,C 180,E1 -11780.822,E2 -11780.822} C_VEL
LIN {X 0,Y 389.595,Z 596.953,A -85,B 0,C 180,E1 -11781.684,E2 -11781.684} C_VEL
LIN {X 0,Y 386.764,Z 597.305,A -85,B 0,C 180,E1 -11783.087,E2 -11783.087} C_VEL
LIN {X 0,Y 384.312,Z 597.614,A -85,B 0,C 180,E1 -11784.22,E2 -11784.22} C_VEL
LIN {X 0,Y 383.217,Z 597.747,A -85,B 0,C 180,E1 -11785.096,E2 -11785.096} C_VEL
LIN {X 0,Y 383.107,Z 597.759,A -85,B 0,C 180,E1 -11785.393,E2 -11785.393} C_VEL
LIN {X 0,Y 383.389,Z 597.725,A -85,B 0,C 180,E1 -11787.9,E2 -11787.9} C_VEL
LIN {X 0,Y 383.519,Z 597.709,A -85,B 0,C 180,E1 -11790.001,E2 -11790.001} C_VEL
LIN {X 0,Y 383.253,Z 597.742,A -85,B 0,C 180,E1 -11793.155,E2 -11793.155} C_VEL
LIN {X 0,Y 383.29,Z 597.74,A -85,B 0,C 180,E1 -11796.317,E2 -11796.317} C_VEL
LIN {X 0,Y 383.262,Z 597.744,A -85,B 0,C 180,E1 -11798.437,E2 -11798.437} C_VEL
LIN {X 0,Y 383.1,Z 597.76,A -85,B 0,C 180,E1 -11801.643,E2 -11801.643} C_VEL
LIN {X 0,Y 383.113,Z 597.765,A -85,B 0,C 180,E1 -11804.883,E2 -11804.883} C_VEL
LIN {X 0,Y 383.066,Z 597.765,A -85,B 0,C 180,E1 -11808.174,E2 -11808.174} C_VEL
LIN {X 0,Y 382.996,Z 597.774,A -85,B 0,C 180,E1 -11811.532,E2 -11811.532} C_VEL
LIN {X 0,Y 383.056,Z 597.773,A -85,B 0,C 180,E1 -11814.961,E2 -11814.961} C_VEL
LIN {X 0,Y 383.033,Z 597.769,A -85,B 0,C 180,E1 -11818.271,E2 -11818.271} C_VEL
LIN {X 0,Y 383.013,Z 597.771,A -85,B 0,C 180,E1 -11822.15,E2 -11822.15} C_VEL
LIN {X 0,Y 383.022,Z 597.772,A -85,B 0,C 180,E1 -11824.669,E2 -11824.669} C_VEL
LIN {X 0,Y 383.004,Z 597.773,A -85,B 0,C 180,E1 -11827.905,E2 -11827.905} C_VEL
LIN {X 0,Y 382.989,Z 597.781,A -85,B 0,C 180,E1 -11831.348,E2 -11831.348} C_VEL
LIN {X 0,Y 383,Z 597.773,A -85,B 0,C 180,E1 -11834.304,E2 -11834.304} C_VEL
LIN {X 0,Y 383.014,Z 597.776,A -85,B 0,C 180,E1 -11837.241,E2 -11837.241} C_VEL
LIN {X 0,Y 383.018,Z 597.77,A -85,B 0,C 180,E1 -11840.414,E2 -11840.414} C_VEL
LIN {X 0,Y 383.029,Z 597.771,A -85,B 0,C 180,E1 -11844.045,E2 -11844.045} C_VEL
LIN {X 0,Y 383.01,Z 597.779,A -85,B 0,C 180,E1 -11847.574,E2 -11847.574} C_VEL
LIN {X 0,Y 382.997,Z 597.774,A -85,B 0,C 180,E1 -11850.301,E2 -11850.301} C_VEL
LIN {X 0,Y 383.061,Z 597.765,A -85,B 0,C 180,E1 -11852.699,E2 -11852.699} C_VEL
LIN {X 0,Y 383.056,Z 597.766,A -85,B 0,C 180,E1 -11855.04,E2 -11855.04} C_VEL
LIN {X 0,Y 382.997,Z 597.774,A -85,B 0,C 180,E1 -11858.469,E2 -11858.469} C_VEL
LIN {X 0,Y 383.094,Z 597.768,A -85,B 0,C 180,E1 -11861.828,E2 -11861.828} C_VEL
LIN {X 0,Y 383.116,Z 597.758,A -85,B 0,C 180,E1 -11865.119,E2 -11865.119} C_VEL
LIN {X 0,Y 383.102,Z 597.763,A -85,B 0,C 180,E1 -11868.358,E2 -11868.358} C_VEL
LIN {X 0,Y 383.269,Z 597.746,A -85,B 0,C 180,E1 -11871.976,E2 -11871.976} C_VEL
LIN {X 0,Y 383.202,Z 597.748,A -85,B 0,C 180,E1 -11874.739,E2 -11874.739} C_VEL
LIN {X 0,Y 383.391,Z 597.728,A -85,B 0,C 180,E1 -11877.899,E2 -11877.899} C_VEL
LIN {X 0,Y 383.523,Z 597.712,A -85,B 0,C 180,E1 -11880,E2 -11880} C_VEL
LIN {X 0,Y 383.252,Z 597.741,A -85,B 0,C 180,E1 -11883.154,E2 -11883.154} C_VEL
LIN {X 0,Y 383.289,Z 597.744,A -85,B 0,C 180,E1 -11886.316,E2 -11886.316} C_VEL
LIN {X 0,Y 383.157,Z 597.753,A -85,B 0,C 180,E1 -11889.502,E2 -11889.502} C_VEL
LIN {X 0,Y 383.131,Z 597.756,A -85,B 0,C 180,E1 -11893.536,E2 -11893.536} C_VEL
LIN {X 0,Y 383.1,Z 597.762,A -85,B 0,C 180,E1 -11897.069,E2 -11897.069} C_VEL
LIN {X 0,Y 383.035,Z 597.775,A -85,B 0,C 180,E1 -11900.647,E2 -11900.647} C_VEL
LIN {X 0,Y 383.032,Z 597.769,A -85,B 0,C 180,E1 -11903.808,E2 -11903.808} C_VEL
LIN {X 0,Y 383.086,Z 597.763,A -85,B 0,C 180,E1 -11906.123,E2 -11906.123} C_VEL
LIN {X 0,Y 383.046,Z 597.771,A -85,B 0,C 180,E1 -11908.492,E2 -11908.492} C_VEL
LIN {X 0,Y 383.015,Z 597.772,A -85,B 0,C 180,E1 -11912.149,E2 -11912.149} C_VEL
LIN {X 0,Y 383.024,Z 597.775,A -85,B 0,C 180,E1 -11914.668,E2 -11914.668} C_VEL
LIN {X 0,Y 383.004,Z 597.772,A -85,B 0,C 180,E1 -11917.903,E2 -11917.903} C_VEL
LIN {X 0,Y 382.989,Z 597.777,A -85,B 0,C 180,E1 -11921.347,E2 -11921.347} C_VEL
LIN {X 0,Y 383.001,Z 597.773,A -85,B 0,C 180,E1 -11924.303,E2 -11924.303} C_VEL
LIN {X 0,Y 383.015,Z 597.776,A -85,B 0,C 180,E1 -11927.24,E2 -11927.24} C_VEL
LIN {X 0,Y 383.02,Z 597.771,A -85,B 0,C 180,E1 -11930.413,E2 -11930.413} C_VEL
LIN {X 0,Y 383.03,Z 597.769,A -85,B 0,C 180,E1 -11934.044,E2 -11934.044} C_VEL
LIN {X 0,Y 382.992,Z 597.779,A -85,B 0,C 180,E1 -11937.577,E2 -11937.577} C_VEL
LIN {X 0,Y 383.047,Z 597.925,A -85,B 0,C 180,E1 -11939.694,E2 -11939.694} C_VEL
LIN {X 0,Y 386.266,Z 612.714,A -85,B 0,C 180,E1 -11943.068,E2 -11943.068} C_VEL
LIN {X 0,Y 387.083,Z 617.721,A -85,B 0,C 180,E1 -11944.166,E2 -11944.166} C_VEL
LIN {X 0,Y 385.961,Z 631.408,A -85,B 0,C 180,E1 -11946.951,E2 -11946.951} C_VEL
LIN {X 0,Y 385.004,Z 643.711,A -85,B 0,C 180,E1 -11949.426,E2 -11949.426} C_VEL
LIN {X 0,Y 389.436,Z 676.185,A -85,B 0,C 180,E1 -11950.334,E2 -11950.334} C_VEL
LIN {X 0,Y 388.091,Z 752.895,A -85,B 0,C 180,E1 -11951.898,E2 -11951.898} C_VEL
LIN {X 0,Y 387.527,Z 766.456,A -85,B 0,C 180,E1 -11952.383,E2 -11952.383} C_VEL
LIN {X 0,Y 386.752,Z 778.826,A -85,B 0,C 180,E1 -11953.028,E2 -11953.028} C_VEL
LIN {X 0,Y 385.908,Z 790.753,A -85,B 0,C 180,E1 -11953.874,E2 -11953.874} C_VEL
LIN {X 0,Y 385.049,Z 802.25,A -85,B 0,C 180,E1 -11954.923,E2 -11954.923} C_VEL
LIN {X 0,Y 384.29,Z 812.15,A -85,B 0,C 180,E1 -11956.048,E2 -11956.048} C_VEL
LIN {X 0,Y 383.525,Z 821.134,A -85,B 0,C 180,E1 -11957.296,E2 -11957.296} C_VEL
LIN {X 0,Y 382.735,Z 830.34,A -85,B 0,C 180,E1 -11958.882,E2 -11958.882} C_VEL
LIN {X 0,Y 382.237,Z 837.76,A -85,B 0,C 180,E1 -11960.474,E2 -11960.474} C_VEL
LIN {X 0,Y 381.918,Z 843.689,A -85,B 0,C 180,E1 -11962.066,E2 -11962.066} C_VEL
LIN {X 0,Y 381.741,Z 848.696,A -85,B 0,C 180,E1 -11963.808,E2 -11963.808} C_VEL
LIN {X 0,Y 381.724,Z 850.769,A -85,B 0,C 180,E1 -11964.717,E2 -11964.717} C_VEL
LIN {X 0,Y 381.663,Z 852.751,A -85,B 0,C 180,E1 -11965.775,E2 -11965.775} C_VEL
LIN {X 0,Y 381.662,Z 854.306,A -85,B 0,C 180,E1 -11966.832,E2 -11966.832} C_VEL
LIN {X 0,Y 381.776,Z 855.397,A -85,B 0,C 180,E1 -11967.889,E2 -11967.889} C_VEL
LIN {X 0,Y 381.732,Z 856.057,A -85,B 0,C 180,E1 -11968.944,E2 -11968.944} C_VEL
LIN {X 0,Y 381.725,Z 856.316,A -85,B 0,C 180,E1 -11969.999,E2 -11969.999} C_VEL
LIN {X 0,Y 381.732,Z 856.167,A -85,B 0,C 180,E1 -11971.054,E2 -11971.054} C_VEL
LIN {X 0,Y 381.758,Z 855.567,A -85,B 0,C 180,E1 -11972.109,E2 -11972.109} C_VEL
LIN {X 0,Y 381.656,Z 853.125,A -85,B 0,C 180,E1 -11974.223,E2 -11974.223} C_VEL
LIN {X 0,Y 381.693,Z 849.435,A -85,B 0,C 180,E1 -11976.126,E2 -11976.126} C_VEL
LIN {X 0,Y 381.915,Z 844.482,A -85,B 0,C 180,E1 -11977.932,E2 -11977.932} C_VEL
LIN {X 0,Y 382.363,Z 837.812,A -85,B 0,C 180,E1 -11979.788,E2 -11979.788} C_VEL
LIN {X 0,Y 382.888,Z 830.533,A -85,B 0,C 180,E1 -11981.379,E2 -11981.379} C_VEL
LIN {X 0,Y 383.775,Z 821.482,A -85,B 0,C 180,E1 -11982.962,E2 -11982.962} C_VEL
LIN {X 0,Y 384.616,Z 811.906,A -85,B 0,C 180,E1 -11984.324,E2 -11984.324} C_VEL
LIN {X 0,Y 385.516,Z 802.042,A -85,B 0,C 180,E1 -11985.462,E2 -11985.462} C_VEL
LIN {X 0,Y 386.474,Z 790.773,A -85,B 0,C 180,E1 -11986.506,E2 -11986.506} C_VEL
LIN {X 0,Y 387.466,Z 778.219,A -85,B 0,C 180,E1 -11987.413,E2 -11987.413} C_VEL
LIN {X 0,Y 388.381,Z 765.517,A -85,B 0,C 180,E1 -11988.085,E2 -11988.085} C_VEL
LIN {X 0,Y 389.079,Z 752.351,A -85,B 0,C 180,E1 -11988.563,E2 -11988.563} C_VEL
LIN {X 0,Y 390.039,Z 703.578,A -85,B 0,C 180,E1 -11989.596,E2 -11989.596} C_VEL
LIN {X 0,Y 390.534,Z 675.762,A -85,B 0,C 180,E1 -11990.181,E2 -11990.181} C_VEL
LIN {X 0,Y 387.472,Z 652.97,A -85,B 0,C 180,E1 -11990.886,E2 -11990.886} C_VEL
LIN {X 0,Y 385.453,Z 641.435,A -85,B 0,C 180,E1 -11991.292,E2 -11991.292} C_VEL
LIN {X 0,Y 386.942,Z 624.727,A -85,B 0,C 180,E1 -11994.749,E2 -11994.749} C_VEL
LIN {X 0,Y 387.46,Z 618.367,A -85,B 0,C 180,E1 -11996.094,E2 -11996.094} C_VEL
LIN {X 0,Y 385.406,Z 607.685,A -85,B 0,C 180,E1 -11998.635,E2 -11998.635} C_VEL
LIN {X 0,Y 382.986,Z 597.785,A -85,B 0,C 180,E1 -12001.185,E2 -12001.185} C_VEL
LIN {X 0,Y 383.015,Z 597.777,A -85,B 0,C 180,E1 -12004.667,E2 -12004.667} C_VEL
LIN {X 0,Y 383,Z 597.777,A -85,B 0,C 180,E1 -12007.903,E2 -12007.903} C_VEL
LIN {X 0,Y 383.009,Z 597.778,A -85,B 0,C 180,E1 -12011.342,E2 -12011.342} C_VEL
LIN {X 0,Y 383.004,Z 597.779,A -85,B 0,C 180,E1 -12014.304,E2 -12014.304} C_VEL
LIN {X 0,Y 383.07,Z 597.768,A -85,B 0,C 180,E1 -12017.248,E2 -12017.248} C_VEL
LIN {X 0,Y 383.017,Z 597.776,A -85,B 0,C 180,E1 -12020.411,E2 -12020.411} C_VEL
LIN {X 0,Y 383.021,Z 597.771,A -85,B 0,C 180,E1 -12024.044,E2 -12024.044} C_VEL
LIN {X 0,Y 383.03,Z 597.771,A -85,B 0,C 180,E1 -12027.852,E2 -12027.852} C_VEL
LIN {X 0,Y 383.057,Z 597.762,A -85,B 0,C 180,E1 -12031.719,E2 -12031.719} C_VEL
LIN {X 0,Y 383.045,Z 597.769,A -85,B 0,C 180,E1 -12035.039,E2 -12035.039} C_VEL
LIN {X 0,Y 382.991,Z 597.779,A -85,B 0,C 180,E1 -12038.469,E2 -12038.469} C_VEL
LIN {X 0,Y 383.081,Z 597.767,A -85,B 0,C 180,E1 -12041.827,E2 -12041.827} C_VEL
LIN {X 0,Y 383.104,Z 597.759,A -85,B 0,C 180,E1 -12045.118,E2 -12045.118} C_VEL
LIN {X 0,Y 383.099,Z 597.764,A -85,B 0,C 180,E1 -12048.358,E2 -12048.358} C_VEL
LIN {X 0,Y 383.295,Z 597.741,A -85,B 0,C 180,E1 -12051.932,E2 -12051.932} C_VEL
LIN {X 0,Y 383.192,Z 597.752,A -85,B 0,C 180,E1 -12054.738,E2 -12054.738} C_VEL
LIN {X 0,Y 383.38,Z 597.73,A -85,B 0,C 180,E1 -12057.899,E2 -12057.899} C_VEL
LIN {X 0,Y 383.513,Z 597.715,A -85,B 0,C 180,E1 -12060,E2 -12060} C_VEL
LIN {X 0,Y 383.246,Z 597.746,A -85,B 0,C 180,E1 -12063.154,E2 -12063.154} C_VEL
LIN {X 0,Y 383.27,Z 597.745,A -85,B 0,C 180,E1 -12066.59,E2 -12066.59} C_VEL
LIN {X 0,Y 383.252,Z 597.749,A -85,B 0,C 180,E1 -12068.436,E2 -12068.436} C_VEL
LIN {X 0,Y 383.139,Z 597.869,A -85,B 0,C 180,E1 -12071.708,E2 -12071.708} C_VEL
LIN {X 0,Y 384.422,Z 604.201,A -85,B 0,C 180,E1 -12073.715,E2 -12073.715} C_VEL
LIN {X 0,Y 389.922,Z 618.071,A -85,B 0,C 180,E1 -12074.424,E2 -12074.424} C_VEL
LIN {X 0,Y 391.495,Z 624.417,A -85,B 0,C 180,E1 -12074.67,E2 -12074.67} C_VEL
LIN {X 0,Y 389.565,Z 710.195,A -85,B 0,C 180,E1 -12076.474,E2 -12076.474} C_VEL
LIN {X 0,Y 389.083,Z 724.099,A -85,B 0,C 180,E1 -12076.99,E2 -12076.99} C_VEL
LIN {X 0,Y 388.382,Z 736.93,A -85,B 0,C 180,E1 -12077.691,E2 -12077.691} C_VEL
LIN {X 0,Y 387.585,Z 749.599,A -85,B 0,C 180,E1 -12078.638,E2 -12078.638} C_VEL
LIN {X 0,Y 386.749,Z 760.307,A -85,B 0,C 180,E1 -12079.66,E2 -12079.66} C_VEL
LIN {X 0,Y 385.754,Z 770.041,A -85,B 0,C 180,E1 -12080.81,E2 -12080.81} C_VEL
LIN {X 0,Y 384.807,Z 779.951,A -85,B 0,C 180,E1 -12082.273,E2 -12082.273} C_VEL
LIN {X 0,Y 383.934,Z 788.099,A -85,B 0,C 180,E1 -12083.761,E2 -12083.761} C_VEL
LIN {X 0,Y 383.264,Z 795.447,A -85,B 0,C 180,E1 -12085.46,E2 -12085.46} C_VEL
LIN {X 0,Y 382.619,Z 801.759,A -85,B 0,C 180,E1 -12087.336,E2 -12087.336} C_VEL
LIN {X 0,Y 382.178,Z 806.316,A -85,B 0,C 180,E1 -12089.164,E2 -12089.164} C_VEL
LIN {X 0,Y 381.896,Z 809.495,A -85,B 0,C 180,E1 -12091.016,E2 -12091.016} C_VEL
LIN {X 0,Y 381.718,Z 810.936,A -85,B 0,C 180,E1 -12092.272,E2 -12092.272} C_VEL
LIN {X 0,Y 381.591,Z 811.945,A -85,B 0,C 180,E1 -12094.028,E2 -12094.028} C_VEL
LIN {X 0,Y 381.578,Z 811.778,A -85,B 0,C 180,E1 -12095.867,E2 -12095.867} C_VEL
LIN {X 0,Y 381.641,Z 810.453,A -85,B 0,C 180,E1 -12097.643,E2 -12097.643} C_VEL
LIN {X 0,Y 381.845,Z 808.026,A -85,B 0,C 180,E1 -12099.376,E2 -12099.376} C_VEL
LIN {X 0,Y 382.108,Z 804.545,A -85,B 0,C 180,E1 -12101.055,E2 -12101.055} C_VEL
LIN {X 0,Y 382.433,Z 799.525,A -85,B 0,C 180,E1 -12102.84,E2 -12102.84} C_VEL
LIN {X 0,Y 382.988,Z 793.092,A -85,B 0,C 180,E1 -12104.579,E2 -12104.579} C_VEL
LIN {X 0,Y 383.529,Z 786.033,A -85,B 0,C 180,E1 -12106.097,E2 -12106.097} C_VEL
LIN {X 0,Y 384.369,Z 777.289,A -85,B 0,C 180,E1 -12107.614,E2 -12107.614} C_VEL
LIN {X 0,Y 385.116,Z 767.924,A -85,B 0,C 180,E1 -12108.933,E2 -12108.933} C_VEL
LIN {X 0,Y 385.984,Z 756.859,A -85,B 0,C 180,E1 -12110.179,E2 -12110.179} C_VEL
LIN {X 0,Y 386.784,Z 745.039,A -85,B 0,C 180,E1 -12111.237,E2 -12111.237} C_VEL
LIN {X 0,Y 387.495,Z 733.268,A -85,B 0,C 180,E1 -12112.043,E2 -12112.043} C_VEL
LIN {X 0,Y 388.04,Z 719.746,A -85,B 0,C 180,E1 -12112.728,E2 -12112.728} C_VEL
LIN {X 0,Y 388.462,Z 706.626,A -85,B 0,C 180,E1 -12113.162,E2 -12113.162} C_VEL
LIN {X 0,Y 389.903,Z 622.846,A -85,B 0,C 180,E1 -12114.855,E2 -12114.855} C_VEL
LIN {X 0,Y 387.449,Z 612.514,A -85,B 0,C 180,E1 -12115.194,E2 -12115.194} C_VEL
LIN {X 0,Y 383.801,Z 601.563,A -85,B 0,C 180,E1 -12115.631,E2 -12115.631} C_VEL
LIN {X 0,Y 383.055,Z 597.769,A -85,B 0,C 180,E1 -12116.741,E2 -12116.741} C_VEL
LIN {X 0,Y 382.988,Z 597.778,A -85,B 0,C 180,E1 -12120.301,E2 -12120.301} C_VEL
LIN {X 0,Y 383.077,Z 597.77,A -85,B 0,C 180,E1 -12124.022,E2 -12124.022} C_VEL
LIN {X 0,Y 383.011,Z 597.771,A -85,B 0,C 180,E1 -12127.337,E2 -12127.337} C_VEL
LIN {X 0,Y 383.07,Z 597.765,A -85,B 0,C 180,E1 -12130.718,E2 -12130.718} C_VEL
LIN {X 0,Y 383.08,Z 597.767,A -85,B 0,C 180,E1 -12134.028,E2 -12134.028} C_VEL
LIN {X 0,Y 383.141,Z 597.755,A -85,B 0,C 180,E1 -12137.285,E2 -12137.285} C_VEL
LIN {X 0,Y 383.175,Z 597.753,A -85,B 0,C 180,E1 -12140.833,E2 -12140.833} C_VEL
LIN {X 0,Y 383.288,Z 597.737,A -85,B 0,C 180,E1 -12143.685,E2 -12143.685} C_VEL
LIN {X 0,Y 383.107,Z 597.759,A -85,B 0,C 180,E1 -12145.393,E2 -12145.393} C_VEL
LIN {X 0,Y 382.462,Z 597.844,A -85,B 0,C 180,E1 -12146.271,E2 -12146.271} C_VEL
LIN {X 0,Y 379.884,Z 598.166,A -85,B 0,C 180,E1 -12147.705,E2 -12147.705} C_VEL
LIN {X 0,Y 376.871,Z 598.54,A -85,B 0,C 180,E1 -12149.453,E2 -12149.453} C_VEL
LIN {X 0,Y 376.475,Z 598.587,A -85,B 0,C 180,E1 -12150.053,E2 -12150.053} C_VEL
LIN {X 0,Y 376.191,Z 598.622,A -85,B 0,C 180,E1 -12153.214,E2 -12153.214} C_VEL
LIN {X 0,Y 376.249,Z 598.618,A -85,B 0,C 180,E1 -12156.436,E2 -12156.436} C_VEL
LIN {X 0,Y 376.207,Z 598.625,A -85,B 0,C 180,E1 -12158.596,E2 -12158.596} C_VEL
LIN {X 0,Y 376.052,Z 598.638,A -85,B 0,C 180,E1 -12161.864,E2 -12161.864} C_VEL
LIN {X 0,Y 376.061,Z 598.64,A -85,B 0,C 180,E1 -12165.168,E2 -12165.168} C_VEL
LIN {X 0,Y 376.012,Z 598.646,A -85,B 0,C 180,E1 -12168.528,E2 -12168.528} C_VEL
LIN {X 0,Y 375.966,Z 598.649,A -85,B 0,C 180,E1 -12171.955,E2 -12171.955} C_VEL
LIN {X 0,Y 376.01,Z 598.646,A -85,B 0,C 180,E1 -12175.462,E2 -12175.462} C_VEL
LIN {X 0,Y 375.965,Z 598.656,A -85,B 0,C 180,E1 -12179.081,E2 -12179.081} C_VEL
LIN {X 0,Y 375.953,Z 598.654,A -85,B 0,C 180,E1 -12182.829,E2 -12182.829} C_VEL
LIN {X 0,Y 375.961,Z 598.654,A -85,B 0,C 180,E1 -12185.416,E2 -12185.416} C_VEL
LIN {X 0,Y 375.978,Z 598.647,A -85,B 0,C 180,E1 -12188.271,E2 -12188.271} C_VEL
LIN {X 0,Y 375.939,Z 598.656,A -85,B 0,C 180,E1 -12191.602,E2 -12191.602} C_VEL
LIN {X 0,Y 375.956,Z 598.656,A -85,B 0,C 180,E1 -12195.265,E2 -12195.265} C_VEL
LIN {X 0,Y 375.944,Z 598.655,A -85,B 0,C 180,E1 -12199.134,E2 -12199.134} C_VEL
LIN {X 0,Y 375.967,Z 598.651,A -85,B 0,C 180,E1 -12201.912,E2 -12201.912} C_VEL
LIN {X 0,Y 375.984,Z 598.651,A -85,B 0,C 180,E1 -12205.333,E2 -12205.333} C_VEL
LIN {X 0,Y 375.962,Z 598.649,A -85,B 0,C 180,E1 -12208.439,E2 -12208.439} C_VEL
LIN {X 0,Y 376.001,Z 598.647,A -85,B 0,C 180,E1 -12212.142,E2 -12212.142} C_VEL
LIN {X 0,Y 376.01,Z 598.644,A -85,B 0,C 180,E1 -12214.539,E2 -12214.539} C_VEL
LIN {X 0,Y 375.962,Z 598.653,A -85,B 0,C 180,E1 -12218.046,E2 -12218.046} C_VEL
LIN {X 0,Y 376.029,Z 598.644,A -85,B 0,C 180,E1 -12221.474,E2 -12221.474} C_VEL
LIN {X 0,Y 376.064,Z 598.637,A -85,B 0,C 180,E1 -12224.833,E2 -12224.833} C_VEL
LIN {X 0,Y 376.055,Z 598.643,A -85,B 0,C 180,E1 -12228.137,E2 -12228.137} C_VEL
LIN {X 0,Y 376.224,Z 598.622,A -85,B 0,C 180,E1 -12231.919,E2 -12231.919} C_VEL
LIN {X 0,Y 376.175,Z 598.624,A -85,B 0,C 180,E1 -12234.64,E2 -12234.64} C_VEL
LIN {X 0,Y 376.357,Z 598.604,A -85,B 0,C 180,E1 -12237.86,E2 -12237.86} C_VEL
LIN {X 0,Y 376.493,Z 598.588,A -85,B 0,C 180,E1 -12240,E2 -12240} C_VEL
LIN {X 0,Y 376.19,Z 598.621,A -85,B 0,C 180,E1 -12243.213,E2 -12243.213} C_VEL
LIN {X 0,Y 376.247,Z 598.619,A -85,B 0,C 180,E1 -12246.435,E2 -12246.435} C_VEL
LIN {X 0,Y 376.125,Z 598.63,A -85,B 0,C 180,E1 -12249.681,E2 -12249.681} C_VEL
LIN {X 0,Y 376.095,Z 598.633,A -85,B 0,C 180,E1 -12253.658,E2 -12253.658} C_VEL
LIN {X 0,Y 376.038,Z 598.64,A -85,B 0,C 180,E1 -12257.4,E2 -12257.4} C_VEL
LIN {X 0,Y 375.984,Z 598.651,A -85,B 0,C 180,E1 -12260.832,E2 -12260.832} C_VEL
LIN {X 0,Y 375.996,Z 598.648,A -85,B 0,C 180,E1 -12264.282,E2 -12264.282} C_VEL
LIN {X 0,Y 376.026,Z 598.648,A -85,B 0,C 180,E1 -12266.652,E2 -12266.652} C_VEL
LIN {X 0,Y 375.976,Z 598.651,A -85,B 0,C 180,E1 -12269.079,E2 -12269.079} C_VEL
LIN {X 0,Y 375.955,Z 598.657,A -85,B 0,C 180,E1 -12272.828,E2 -12272.828} C_VEL
LIN {X 0,Y 375.963,Z 598.651,A -85,B 0,C 180,E1 -12275.415,E2 -12275.415} C_VEL
LIN {X 0,Y 375.979,Z 598.648,A -85,B 0,C 180,E1 -12278.27,E2 -12278.27} C_VEL
LIN {X 0,Y 375.94,Z 598.653,A -85,B 0,C 180,E1 -12281.6,E2 -12281.6} C_VEL
LIN {X 0,Y 375.958,Z 598.654,A -85,B 0,C 180,E1 -12285.264,E2 -12285.264} C_VEL
LIN {X 0,Y 375.945,Z 598.658,A -85,B 0,C 180,E1 -12289.132,E2 -12289.132} C_VEL
LIN {X 0,Y 375.969,Z 598.649,A -85,B 0,C 180,E1 -12291.911,E2 -12291.911} C_VEL
LIN {X 0,Y 375.985,Z 598.653,A -85,B 0,C 180,E1 -12295.332,E2 -12295.332} C_VEL
LIN {X 0,Y 375.963,Z 598.653,A -85,B 0,C 180,E1 -12298.437,E2 -12298.437} C_VEL
LIN {X 0,Y 375.998,Z 598.837,A -85,B 0,C 180,E1 -12299.411,E2 -12299.411} C_VEL
LIN {X 0,Y 378.771,Z 611.451,A -85,B 0,C 180,E1 -12302.362,E2 -12302.362} C_VEL
LIN {X 0,Y 380.07,Z 618.488,A -85,B 0,C 180,E1 -12303.948,E2 -12303.948} C_VEL
LIN {X 0,Y 379.473,Z 626.957,A -85,B 0,C 180,E1 -12305.716,E2 -12305.716} C_VEL
LIN {X 0,Y 378.105,Z 643.375,A -85,B 0,C 180,E1 -12309.087,E2 -12309.087} C_VEL
LIN {X 0,Y 382.617,Z 677.393,A -85,B 0,C 180,E1 -12310.048,E2 -12310.048} C_VEL
LIN {X 0,Y 381.227,Z 753.129,A -85,B 0,C 180,E1 -12311.63,E2 -12311.63} C_VEL
LIN {X 0,Y 380.666,Z 766.479,A -85,B 0,C 180,E1 -12312.124,E2 -12312.124} C_VEL
LIN {X 0,Y 379.85,Z 778.719,A -85,B 0,C 180,E1 -12312.779,E2 -12312.779} C_VEL
LIN {X 0,Y 379.08,Z 789.784,A -85,B 0,C 180,E1 -12313.576,E2 -12313.576} C_VEL
LIN {X 0,Y 378.128,Z 801.377,A -85,B 0,C 180,E1 -12314.641,E2 -12314.641} C_VEL
LIN {X 0,Y 377.307,Z 811.883,A -85,B 0,C 180,E1 -12315.851,E2 -12315.851} C_VEL
LIN {X 0,Y 376.526,Z 820.424,A -85,B 0,C 180,E1 -12317.056,E2 -12317.056} C_VEL
LIN {X 0,Y 375.732,Z 829.698,A -85,B 0,C 180,E1 -12318.672,E2 -12318.672} C_VEL
LIN {X 0,Y 375.187,Z 837.161,A -85,B 0,C 180,E1 -12320.293,E2 -12320.293} C_VEL
LIN {X 0,Y 374.86,Z 843.134,A -85,B 0,C 180,E1 -12321.916,E2 -12321.916} C_VEL
LIN {X 0,Y 374.667,Z 848.476,A -85,B 0,C 180,E1 -12323.814,E2 -12323.814} C_VEL
LIN {X 0,Y 374.591,Z 852.272,A -85,B 0,C 180,E1 -12325.695,E2 -12325.695} C_VEL
LIN {X 0,Y 374.568,Z 853.84,A -85,B 0,C 180,E1 -12326.772,E2 -12326.772} C_VEL
LIN {X 0,Y 374.689,Z 854.954,A -85,B 0,C 180,E1 -12327.849,E2 -12327.849} C_VEL
LIN {X 0,Y 374.664,Z 855.626,A -85,B 0,C 180,E1 -12328.924,E2 -12328.924} C_VEL
LIN {X 0,Y 374.655,Z 855.894,A -85,B 0,C 180,E1 -12329.999,E2 -12329.999} C_VEL
LIN {X 0,Y 374.663,Z 855.758,A -85,B 0,C 180,E1 -12331.074,E2 -12331.074} C_VEL
LIN {X 0,Y 374.673,Z 855.171,A -85,B 0,C 180,E1 -12332.149,E2 -12332.149} C_VEL
LIN {X 0,Y 374.58,Z 852.747,A -85,B 0,C 180,E1 -12334.303,E2 -12334.303} C_VEL
LIN {X 0,Y 374.592,Z 849.452,A -85,B 0,C 180,E1 -12336.078,E2 -12336.078} C_VEL
LIN {X 0,Y 374.767,Z 845.76,A -85,B 0,C 180,E1 -12337.542,E2 -12337.542} C_VEL
LIN {X 0,Y 375.149,Z 839.608,A -85,B 0,C 180,E1 -12339.433,E2 -12339.433} C_VEL
LIN {X 0,Y 375.666,Z 832.85,A -85,B 0,C 180,E1 -12341.054,E2 -12341.054} C_VEL
LIN {X 0,Y 376.527,Z 824.481,A -85,B 0,C 180,E1 -12342.668,E2 -12342.668} C_VEL
LIN {X 0,Y 377.322,Z 815.954,A -85,B 0,C 180,E1 -12344.011,E2 -12344.011} C_VEL
LIN {X 0,Y 378.274,Z 805.501,A -85,B 0,C 180,E1 -12345.351,E2 -12345.351} C_VEL
LIN {X 0,Y 379.418,Z 793.759,A -85,B 0,C 180,E1 -12346.545,E2 -12346.545} C_VEL
LIN {X 0,Y 380.479,Z 782.265,A -85,B 0,C 180,E1 -12347.466,E2 -12347.466} C_VEL
LIN {X 0,Y 381.322,Z 770.508,A -85,B 0,C 180,E1 -12348.189,E2 -12348.189} C_VEL
LIN {X 0,Y 382.233,Z 756.352,A -85,B 0,C 180,E1 -12348.803,E2 -12348.803} C_VEL
LIN {X 0,Y 382.66,Z 743.044,A -85,B 0,C 180,E1 -12349.164,E2 -12349.164} C_VEL
LIN {X 0,Y 383.955,Z 676.268,A -85,B 0,C 180,E1 -12350.581,E2 -12350.581} C_VEL
LIN {X 0,Y 380.847,Z 653.412,A -85,B 0,C 180,E1 -12351.312,E2 -12351.312} C_VEL
LIN {X 0,Y 378.632,Z 640.843,A -85,B 0,C 180,E1 -12351.79,E2 -12351.79} C_VEL
LIN {X 0,Y 380.177,Z 624.921,A -85,B 0,C 180,E1 -12355.161,E2 -12355.161} C_VEL
LIN {X 0,Y 380.544,Z 619.638,A -85,B 0,C 180,E1 -12356.309,E2 -12356.309} C_VEL
LIN {X 0,Y 378.474,Z 609.19,A -85,B 0,C 180,E1 -12358.867,E2 -12358.867} C_VEL
LIN {X 0,Y 375.949,Z 598.66,A -85,B 0,C 180,E1 -12361.64,E2 -12361.64} C_VEL
LIN {X 0,Y 375.955,Z 598.655,A -85,B 0,C 180,E1 -12365.414,E2 -12365.414} C_VEL
LIN {X 0,Y 375.974,Z 598.655,A -85,B 0,C 180,E1 -12368.27,E2 -12368.27} C_VEL
LIN {X 0,Y 375.956,Z 598.657,A -85,B 0,C 180,E1 -12371.604,E2 -12371.604} C_VEL
LIN {X 0,Y 375.976,Z 598.653,A -85,B 0,C 180,E1 -12375.259,E2 -12375.259} C_VEL
LIN {X 0,Y 375.984,Z 598.652,A -85,B 0,C 180,E1 -12378.389,E2 -12378.389} C_VEL
LIN {X 0,Y 375.962,Z 598.652,A -85,B 0,C 180,E1 -12381.911,E2 -12381.911} C_VEL
LIN {X 0,Y 375.974,Z 598.649,A -85,B 0,C 180,E1 -12385.332,E2 -12385.332} C_VEL
LIN {X 0,Y 375.971,Z 598.649,A -85,B 0,C 180,E1 -12388.439,E2 -12388.439} C_VEL
LIN {X 0,Y 375.996,Z 598.645,A -85,B 0,C 180,E1 -12392.141,E2 -12392.141} C_VEL
LIN {X 0,Y 375.999,Z 598.646,A -85,B 0,C 180,E1 -12394.538,E2 -12394.538} C_VEL
LIN {X 0,Y 375.96,Z 598.653,A -85,B 0,C 180,E1 -12398.045,E2 -12398.045} C_VEL
LIN {X 0,Y 376.016,Z 598.645,A -85,B 0,C 180,E1 -12401.473,E2 -12401.473} C_VEL
LIN {X 0,Y 376.051,Z 598.639,A -85,B 0,C 180,E1 -12404.832,E2 -12404.832} C_VEL
LIN {X 0,Y 376.051,Z 598.64,A -85,B 0,C 180,E1 -12408.136,E2 -12408.136} C_VEL
LIN {X 0,Y 376.249,Z 598.619,A -85,B 0,C 180,E1 -12411.877,E2 -12411.877} C_VEL
LIN {X 0,Y 376.164,Z 598.627,A -85,B 0,C 180,E1 -12414.64,E2 -12414.64} C_VEL
LIN {X 0,Y 376.346,Z 598.606,A -85,B 0,C 180,E1 -12417.859,E2 -12417.859} C_VEL
LIN {X 0,Y 376.482,Z 598.591,A -85,B 0,C 180,E1 -12420,E2 -12420} C_VEL
LIN {X 0,Y 376.184,Z 598.626,A -85,B 0,C 180,E1 -12423.213,E2 -12423.213} C_VEL
LIN {X 0,Y 376.235,Z 598.622,A -85,B 0,C 180,E1 -12426.579,E2 -12426.579} C_VEL
LIN {X 0,Y 376.197,Z 598.627,A -85,B 0,C 180,E1 -12428.595,E2 -12428.595} C_VEL
LIN {X 0,Y 376.069,Z 598.699,A -85,B 0,C 180,E1 -12431.248,E2 -12431.248} C_VEL
LIN {X 0,Y 377.341,Z 604.759,A -85,B 0,C 180,E1 -12433.223,E2 -12433.223} C_VEL
LIN {X 0,Y 383.786,Z 620.676,A -85,B 0,C 180,E1 -12434.072,E2 -12434.072} C_VEL
LIN {X 0,Y 384.969,Z 626.039,A -85,B 0,C 180,E1 -12434.277,E2 -12434.277} C_VEL
LIN {X 0,Y 382.971,Z 710.897,A -85,B 0,C 180,E1 -12436.103,E2 -12436.103} C_VEL
LIN {X 0,Y 382.474,Z 724.015,A -85,B 0,C 180,E1 -12436.595,E2 -12436.595} C_VEL
LIN {X 0,Y 381.816,Z 736.336,A -85,B 0,C 180,E1 -12437.266,E2 -12437.266} C_VEL
LIN {X 0,Y 381.012,Z 748.156,A -85,B 0,C 180,E1 -12438.136,E2 -12438.136} C_VEL
LIN {X 0,Y 380.07,Z 759.838,A -85,B 0,C 180,E1 -12439.244,E2 -12439.244} C_VEL
LIN {X 0,Y 378.966,Z 770.328,A -85,B 0,C 180,E1 -12440.49,E2 -12440.49} C_VEL
LIN {X 0,Y 378.051,Z 779.335,A -85,B 0,C 180,E1 -12441.827,E2 -12441.827} C_VEL
LIN {X 0,Y 377.192,Z 787.236,A -85,B 0,C 180,E1 -12443.256,E2 -12443.256} C_VEL
LIN {X 0,Y 376.424,Z 794.335,A -85,B 0,C 180,E1 -12444.84,E2 -12444.84} C_VEL
LIN {X 0,Y 375.956,Z 799.254,A -85,B 0,C 180,E1 -12446.199,E2 -12446.199} C_VEL
LIN {X 0,Y 375.443,Z 804.2,A -85,B 0,C 180,E1 -12447.903,E2 -12447.903} C_VEL
LIN {X 0,Y 375.032,Z 808.209,A -85,B 0,C 180,E1 -12449.775,E2 -12449.775} C_VEL
LIN {X 0,Y 374.705,Z 810.864,A -85,B 0,C 180,E1 -12451.68,E2 -12451.68} C_VEL
LIN {X 0,Y 374.564,Z 811.939,A -85,B 0,C 180,E1 -12452.965,E2 -12452.965} C_VEL
LIN {X 0,Y 374.507,Z 812.41,A -85,B 0,C 180,E1 -12454.343,E2 -12454.343} C_VEL
LIN {X 0,Y 374.496,Z 812.017,A -85,B 0,C 180,E1 -12456.202,E2 -12456.202} C_VEL
LIN {X 0,Y 374.609,Z 810.188,A -85,B 0,C 180,E1 -12458.251,E2 -12458.251} C_VEL
LIN {X 0,Y 374.934,Z 806.713,A -85,B 0,C 180,E1 -12460.329,E2 -12460.329} C_VEL
LIN {X 0,Y 375.163,Z 803.016,A -85,B 0,C 180,E1 -12461.885,E2 -12461.885} C_VEL
LIN {X 0,Y 375.617,Z 796.977,A -85,B 0,C 180,E1 -12463.812,E2 -12463.812} C_VEL
LIN {X 0,Y 376.242,Z 790.019,A -85,B 0,C 180,E1 -12465.509,E2 -12465.509} C_VEL
LIN {X 0,Y 377.033,Z 781.203,A -85,B 0,C 180,E1 -12467.219,E2 -12467.219} C_VEL
LIN {X 0,Y 377.852,Z 771.78,A -85,B 0,C 180,E1 -12468.674,E2 -12468.674} C_VEL
LIN {X 0,Y 378.732,Z 761.543,A -85,B 0,C 180,E1 -12469.948,E2 -12469.948} C_VEL
LIN {X 0,Y 379.561,Z 750.571,A -85,B 0,C 180,E1 -12471.048,E2 -12471.048} C_VEL
LIN {X 0,Y 380.338,Z 738.836,A -85,B 0,C 180,E1 -12471.968,E2 -12471.968} C_VEL
LIN {X 0,Y 380.999,Z 725.519,A -85,B 0,C 180,E1 -12472.754,E2 -12472.754} C_VEL
LIN {X 0,Y 381.479,Z 712.443,A -85,B 0,C 180,E1 -12473.286,E2 -12473.286} C_VEL
LIN {X 0,Y 381.824,Z 693.646,A -85,B 0,C 180,E1 -12473.732,E2 -12473.732} C_VEL
LIN {X 0,Y 383.06,Z 623.385,A -85,B 0,C 180,E1 -12475.178,E2 -12475.178} C_VEL
LIN {X 0,Y 380.811,Z 614.14,A -85,B 0,C 180,E1 -12475.489,E2 -12475.489} C_VEL
LIN {X 0,Y 376.643,Z 601.9,A -85,B 0,C 180,E1 -12476.001,E2 -12476.001} C_VEL
LIN {X 0,Y 375.996,Z 598.648,A -85,B 0,C 180,E1 -12476.978,E2 -12476.978} C_VEL
LIN {X 0,Y 375.957,Z 598.65,A -85,B 0,C 180,E1 -12480.921,E2 -12480.921} C_VEL
LIN {X 0,Y 376.003,Z 598.646,A -85,B 0,C 180,E1 -12484.54,E2 -12484.54} C_VEL
LIN {X 0,Y 375.969,Z 598.654,A -85,B 0,C 180,E1 -12488.047,E2 -12488.047} C_VEL
LIN {X 0,Y 376.028,Z 598.642,A -85,B 0,C 180,E1 -12491.476,E2 -12491.476} C_VEL
LIN {X 0,Y 376.059,Z 598.639,A -85,B 0,C 180,E1 -12494.834,E2 -12494.834} C_VEL
LIN {X 0,Y 376.059,Z 598.642,A -85,B 0,C 180,E1 -12498.138,E2 -12498.138} C_VEL
LIN {X 0,Y 376.258,Z 598.614,A -85,B 0,C 180,E1 -12501.878,E2 -12501.878} C_VEL
LIN {X 0,Y 376.172,Z 598.628,A -85,B 0,C 180,E1 -12504.641,E2 -12504.641} C_VEL
LIN {X 0,Y 376.355,Z 598.601,A -85,B 0,C 180,E1 -12507.861,E2 -12507.861} C_VEL
LIN {X 0,Y 376.475,Z 598.587,A -85,B 0,C 180,E1 -12510.053,E2 -12510.053} C_VEL
LIN {X 0,Y 375.617,Z 598.696,A -85,B 0,C 180,E1 -12510.945,E2 -12510.945} C_VEL
LIN {X 0,Y 372.544,Z 599.08,A -85,B 0,C 180,E1 -12512.391,E2 -12512.391} C_VEL
LIN {X 0,Y 370.077,Z 599.388,A -85,B 0,C 180,E1 -12513.561,E2 -12513.561} C_VEL
LIN {X 0,Y 369.086,Z 599.511,A -85,B 0,C 180,E1 -12514.468,E2 -12514.468} C_VEL
LIN {X 0,Y 369.037,Z 599.513,A -85,B 0,C 180,E1 -12514.775,E2 -12514.775} C_VEL
LIN {X 0,Y 369.19,Z 599.493,A -85,B 0,C 180,E1 -12517.659,E2 -12517.659} C_VEL
LIN {X 0,Y 369.024,Z 599.518,A -85,B 0,C 180,E1 -12520.98,E2 -12520.98} C_VEL
LIN {X 0,Y 369.017,Z 599.516,A -85,B 0,C 180,E1 -12524.336,E2 -12524.336} C_VEL
LIN {X 0,Y 369.004,Z 599.516,A -85,B 0,C 180,E1 -12527.769,E2 -12527.769} C_VEL
LIN {X 0,Y 368.932,Z 599.529,A -85,B 0,C 180,E1 -12531.221,E2 -12531.221} C_VEL
LIN {X 0,Y 368.961,Z 599.526,A -85,B 0,C 180,E1 -12534.776,E2 -12534.776} C_VEL
LIN {X 0,Y 368.966,Z 599.526,A -85,B 0,C 180,E1 -12537.204,E2 -12537.204} C_VEL
LIN {X 0,Y 368.933,Z 599.53,A -85,B 0,C 180,E1 -12540.954,E2 -12540.954} C_VEL
LIN {X 0,Y 368.933,Z 599.53,A -85,B 0,C 180,E1 -12545.002,E2 -12545.002} C_VEL
LIN {X 0,Y 368.913,Z 599.529,A -85,B 0,C 180,E1 -12548.641,E2 -12548.641} C_VEL
LIN {X 0,Y 368.885,Z 599.532,A -85,B 0,C 180,E1 -12552.01,E2 -12552.01} C_VEL
LIN {X 0,Y 368.929,Z 599.53,A -85,B 0,C 180,E1 -12555.184,E2 -12555.184} C_VEL
LIN {X 0,Y 368.887,Z 599.531,A -85,B 0,C 180,E1 -12558.178,E2 -12558.178} C_VEL
LIN {X 0,Y 368.912,Z 599.533,A -85,B 0,C 180,E1 -12561.361,E2 -12561.361} C_VEL
LIN {X 0,Y 368.941,Z 599.526,A -85,B 0,C 180,E1 -12565.147,E2 -12565.147} C_VEL
LIN {X 0,Y 368.934,Z 599.526,A -85,B 0,C 180,E1 -12569.047,E2 -12569.047} C_VEL
LIN {X 0,Y 368.985,Z 599.524,A -85,B 0,C 180,E1 -12571.564,E2 -12571.564} C_VEL
LIN {X 0,Y 369.005,Z 599.52,A -85,B 0,C 180,E1 -12574.02,E2 -12574.02} C_VEL
LIN {X 0,Y 368.927,Z 599.531,A -85,B 0,C 180,E1 -12577.605,E2 -12577.605} C_VEL
LIN {X 0,Y 368.972,Z 599.521,A -85,B 0,C 180,E1 -12581.107,E2 -12581.107} C_VEL
LIN {X 0,Y 369.003,Z 599.517,A -85,B 0,C 180,E1 -12584.536,E2 -12584.536} C_VEL
LIN {X 0,Y 369.011,Z 599.522,A -85,B 0,C 180,E1 -12587.907,E2 -12587.907} C_VEL
LIN {X 0,Y 369.171,Z 599.5,A -85,B 0,C 180,E1 -12591.87,E2 -12591.87} C_VEL
LIN {X 0,Y 369.147,Z 599.5,A -85,B 0,C 180,E1 -12594.538,E2 -12594.538} C_VEL
LIN {X 0,Y 369.322,Z 599.48,A -85,B 0,C 180,E1 -12597.819,E2 -12597.819} C_VEL
LIN {X 0,Y 369.462,Z 599.464,A -85,B 0,C 180,E1 -12600,E2 -12600} C_VEL
LIN {X 0,Y 369.322,Z 599.483,A -85,B 0,C 180,E1 -12602.181,E2 -12602.181} C_VEL
LIN {X 0,Y 369.207,Z 599.495,A -85,B 0,C 180,E1 -12606.558,E2 -12606.558} C_VEL
LIN {X 0,Y 369.073,Z 599.509,A -85,B 0,C 180,E1 -12609.868,E2 -12609.868} C_VEL
LIN {X 0,Y 369.043,Z 599.512,A -85,B 0,C 180,E1 -12613.772,E2 -12613.772} C_VEL
LIN {X 0,Y 368.997,Z 599.517,A -85,B 0,C 180,E1 -12617.743,E2 -12617.743} C_VEL
LIN {X 0,Y 368.916,Z 599.528,A -85,B 0,C 180,E1 -12621.221,E2 -12621.221} C_VEL
LIN {X 0,Y 368.961,Z 599.527,A -85,B 0,C 180,E1 -12624.775,E2 -12624.775} C_VEL
LIN {X 0,Y 368.974,Z 599.521,A -85,B 0,C 180,E1 -12627.203,E2 -12627.203} C_VEL
LIN {X 0,Y 368.925,Z 599.526,A -85,B 0,C 180,E1 -12629.69,E2 -12629.69} C_VEL
LIN {X 0,Y 368.903,Z 599.533,A -85,B 0,C 180,E1 -12633.043,E2 -12633.043} C_VEL
LIN {X 0,Y 368.923,Z 599.527,A -85,B 0,C 180,E1 -12636.196,E2 -12636.196} C_VEL
LIN {X 0,Y 368.908,Z 599.535,A -85,B 0,C 180,E1 -12638.953,E2 -12638.953} C_VEL
LIN {X 0,Y 368.886,Z 599.531,A -85,B 0,C 180,E1 -12642.009,E2 -12642.009} C_VEL
LIN {X 0,Y 368.911,Z 599.533,A -85,B 0,C 180,E1 -12645.179,E2 -12645.179} C_VEL
LIN {X 0,Y 368.888,Z 599.531,A -85,B 0,C 180,E1 -12648.177,E2 -12648.177} C_VEL
LIN {X 0,Y 368.914,Z 599.532,A -85,B 0,C 180,E1 -12651.359,E2 -12651.359} C_VEL
LIN {X 0,Y 368.942,Z 599.53,A -85,B 0,C 180,E1 -12655.146,E2 -12655.146} C_VEL
LIN {X 0,Y 368.946,Z 599.707,A -85,B 0,C 180,E1 -12659.116,E2 -12659.116} C_VEL
LIN {X 0,Y 371.626,Z 611.953,A -85,B 0,C 180,E1 -12662.038,E2 -12662.038} C_VEL
LIN {X 0,Y 373.163,Z 620.634,A -85,B 0,C 180,E1 -12664.03,E2 -12664.03} C_VEL
LIN {X 0,Y 371.686,Z 637.044,A -85,B 0,C 180,E1 -12667.486,E2 -12667.486} C_VEL
LIN {X 0,Y 371.189,Z 642.99,A -85,B 0,C 180,E1 -12668.728,E2 -12668.728} C_VEL
LIN {X 0,Y 375.824,Z 677.825,A -85,B 0,C 180,E1 -12669.742,E2 -12669.742} C_VEL
LIN {X 0,Y 374.429,Z 751.911,A -85,B 0,C 180,E1 -12671.32,E2 -12671.32} C_VEL
LIN {X 0,Y 373.847,Z 765.507,A -85,B 0,C 180,E1 -12671.822,E2 -12671.822} C_VEL
LIN {X 0,Y 373.041,Z 777.345,A -85,B 0,C 180,E1 -12672.455,E2 -12672.455} C_VEL
LIN {X 0,Y 372.207,Z 788.673,A -85,B 0,C 180,E1 -12673.264,E2 -12673.264} C_VEL
LIN {X 0,Y 371.192,Z 800.4,A -85,B 0,C 180,E1 -12674.346,E2 -12674.346} C_VEL
LIN {X 0,Y 370.365,Z 810.995,A -85,B 0,C 180,E1 -12675.577,E2 -12675.577} C_VEL
LIN {X 0,Y 369.557,Z 819.647,A -85,B 0,C 180,E1 -12676.807,E2 -12676.807} C_VEL
LIN {X 0,Y 368.89,Z 827.628,A -85,B 0,C 180,E1 -12678.181,E2 -12678.181} C_VEL
LIN {X 0,Y 368.25,Z 835.395,A -85,B 0,C 180,E1 -12679.831,E2 -12679.831} C_VEL
LIN {X 0,Y 367.796,Z 842.553,A -85,B 0,C 180,E1 -12681.759,E2 -12681.759} C_VEL
LIN {X 0,Y 367.638,Z 847.282,A -85,B 0,C 180,E1 -12683.413,E2 -12683.413} C_VEL
LIN {X 0,Y 367.521,Z 850.849,A -85,B 0,C 180,E1 -12685.062,E2 -12685.062} C_VEL
LIN {X 0,Y 367.478,Z 853.363,A -85,B 0,C 180,E1 -12686.71,E2 -12686.71} C_VEL
LIN {X 0,Y 367.604,Z 854.505,A -85,B 0,C 180,E1 -12687.807,E2 -12687.807} C_VEL
LIN {X 0,Y 367.597,Z 855.19,A -85,B 0,C 180,E1 -12688.903,E2 -12688.903} C_VEL
LIN {X 0,Y 367.586,Z 855.47,A -85,B 0,C 180,E1 -12689.999,E2 -12689.999} C_VEL
LIN {X 0,Y 367.596,Z 855.347,A -85,B 0,C 180,E1 -12691.094,E2 -12691.094} C_VEL
LIN {X 0,Y 367.572,Z 854.783,A -85,B 0,C 180,E1 -12692.19,E2 -12692.19} C_VEL
LIN {X 0,Y 367.505,Z 852.381,A -85,B 0,C 180,E1 -12694.386,E2 -12694.386} C_VEL
LIN {X 0,Y 367.49,Z 849.45,A -85,B 0,C 180,E1 -12696.029,E2 -12696.029} C_VEL
LIN {X 0,Y 367.696,Z 845.434,A -85,B 0,C 180,E1 -12697.688,E2 -12697.688} C_VEL
LIN {X 0,Y 368.118,Z 839.316,A -85,B 0,C 180,E1 -12699.615,E2 -12699.615} C_VEL
LIN {X 0,Y 368.677,Z 832.582,A -85,B 0,C 180,E1 -12701.266,E2 -12701.266} C_VEL
LIN {X 0,Y 369.582,Z 824.241,A -85,B 0,C 180,E1 -12702.91,E2 -12702.91} C_VEL
LIN {X 0,Y 370.417,Z 815.776,A -85,B 0,C 180,E1 -12704.278,E2 -12704.278} C_VEL
LIN {X 0,Y 371.435,Z 805.435,A -85,B 0,C 180,E1 -12705.641,E2 -12705.641} C_VEL
LIN {X 0,Y 372.596,Z 793.805,A -85,B 0,C 180,E1 -12706.857,E2 -12706.857} C_VEL
LIN {X 0,Y 373.719,Z 782.437,A -85,B 0,C 180,E1 -12707.792,E2 -12707.792} C_VEL
LIN {X 0,Y 374.604,Z 770.94,A -85,B 0,C 180,E1 -12708.527,E2 -12708.527} C_VEL
LIN {X 0,Y 375.535,Z 757.139,A -85,B 0,C 180,E1 -12709.152,E2 -12709.152} C_VEL
LIN {X 0,Y 376.009,Z 744.788,A -85,B 0,C 180,E1 -12709.517,E2 -12709.517} C_VEL
LIN {X 0,Y 377.458,Z 677.13,A -85,B 0,C 180,E1 -12710.982,E2 -12710.982} C_VEL
LIN {X 0,Y 374.396,Z 654.534,A -85,B 0,C 180,E1 -12711.737,E2 -12711.737} C_VEL
LIN {X 0,Y 371.829,Z 640.464,A -85,B 0,C 180,E1 -12712.269,E2 -12712.269} C_VEL
LIN {X 0,Y 373.638,Z 623.573,A -85,B 0,C 180,E1 -12715.932,E2 -12715.932} C_VEL
LIN {X 0,Y 373.638,Z 620.952,A -85,B 0,C 180,E1 -12716.533,E2 -12716.533} C_VEL
LIN {X 0,Y 371.514,Z 610.222,A -85,B 0,C 180,E1 -12719.229,E2 -12719.229} C_VEL
LIN {X 0,Y 368.936,Z 599.534,A -85,B 0,C 180,E1 -12722.158,E2 -12722.158} C_VEL
LIN {X 0,Y 368.926,Z 599.531,A -85,B 0,C 180,E1 -12725,E2 -12725} C_VEL
LIN {X 0,Y 368.91,Z 599.536,A -85,B 0,C 180,E1 -12728.64,E2 -12728.64} C_VEL
LIN {X 0,Y 368.906,Z 599.536,A -85,B 0,C 180,E1 -12731.817,E2 -12731.817} C_VEL
LIN {X 0,Y 368.95,Z 599.529,A -85,B 0,C 180,E1 -12735.186,E2 -12735.186} C_VEL
LIN {X 0,Y 368.936,Z 599.531,A -85,B 0,C 180,E1 -12738.185,E2 -12738.185} C_VEL
LIN {X 0,Y 368.908,Z 599.53,A -85,B 0,C 180,E1 -12741.358,E2 -12741.358} C_VEL
LIN {X 0,Y 368.93,Z 599.527,A -85,B 0,C 180,E1 -12745.146,E2 -12745.146} C_VEL
LIN {X 0,Y 368.922,Z 599.527,A -85,B 0,C 180,E1 -12749.046,E2 -12749.046} C_VEL
LIN {X 0,Y 368.981,Z 599.515,A -85,B 0,C 180,E1 -12751.564,E2 -12751.564} C_VEL
LIN {X 0,Y 368.95,Z 599.524,A -85,B 0,C 180,E1 -12755.224,E2 -12755.224} C_VEL
LIN {X 0,Y 368.93,Z 599.526,A -85,B 0,C 180,E1 -12758.973,E2 -12758.973} C_VEL
LIN {X 0,Y 368.982,Z 599.521,A -85,B 0,C 180,E1 -12762.257,E2 -12762.257} C_VEL
LIN {X 0,Y 369.029,Z 599.517,A -85,B 0,C 180,E1 -12766.227,E2 -12766.227} C_VEL
LIN {X 0,Y 369.064,Z 599.512,A -85,B 0,C 180,E1 -12770.131,E2 -12770.131} C_VEL
LIN {X 0,Y 369.179,Z 599.498,A -85,B 0,C 180,E1 -12772.342,E2 -12772.342} C_VEL
LIN {X 0,Y 369.137,Z 599.503,A -85,B 0,C 180,E1 -12774.537,E2 -12774.537} C_VEL
LIN {X 0,Y 369.311,Z 599.483,A -85,B 0,C 180,E1 -12777.819,E2 -12777.819} C_VEL
LIN {X 0,Y 369.452,Z 599.467,A -85,B 0,C 180,E1 -12780,E2 -12780} C_VEL
LIN {X 0,Y 369.311,Z 599.483,A -85,B 0,C 180,E1 -12782.181,E2 -12782.181} C_VEL
LIN {X 0,Y 369.206,Z 599.5,A -85,B 0,C 180,E1 -12786.566,E2 -12786.566} C_VEL
LIN {X 0,Y 369.13,Z 599.508,A -85,B 0,C 180,E1 -12788.761,E2 -12788.761} C_VEL
LIN {X 0,Y 369.045,Z 599.561,A -85,B 0,C 180,E1 -12790.77,E2 -12790.77} C_VEL
LIN {X 0,Y 370.362,Z 605.535,A -85,B 0,C 180,E1 -12792.709,E2 -12792.709} C_VEL
LIN {X 0,Y 377.468,Z 622.686,A -85,B 0,C 180,E1 -12793.667,E2 -12793.667} C_VEL
LIN {X 0,Y 378.444,Z 626.064,A -85,B 0,C 180,E1 -12793.82,E2 -12793.82} C_VEL
LIN {X 0,Y 376.396,Z 711.263,A -85,B 0,C 180,E1 -12795.708,E2 -12795.708} C_VEL
LIN {X 0,Y 375.854,Z 724.632,A -85,B 0,C 180,E1 -12796.219,E2 -12796.219} C_VEL
LIN {X 0,Y 375.137,Z 737.484,A -85,B 0,C 180,E1 -12796.94,E2 -12796.94} C_VEL
LIN {X 0,Y 374.368,Z 748.408,A -85,B 0,C 180,E1 -12797.762,E2 -12797.762} C_VEL
LIN {X 0,Y 373.361,Z 760.219,A -85,B 0,C 180,E1 -12798.898,E2 -12798.898} C_VEL
LIN {X 0,Y 372.196,Z 770.684,A -85,B 0,C 180,E1 -12800.158,E2 -12800.158} C_VEL
LIN {X 0,Y 371.206,Z 779.851,A -85,B 0,C 180,E1 -12801.542,E2 -12801.542} C_VEL
LIN {X 0,Y 370.168,Z 788.727,A -85,B 0,C 180,E1 -12803.201,E2 -12803.201} C_VEL
LIN {X 0,Y 369.415,Z 795.333,A -85,B 0,C 180,E1 -12804.743,E2 -12804.743} C_VEL
LIN {X 0,Y 368.822,Z 801.048,A -85,B 0,C 180,E1 -12806.418,E2 -12806.418} C_VEL
LIN {X 0,Y 368.387,Z 804.993,A -85,B 0,C 180,E1 -12807.866,E2 -12807.866} C_VEL
LIN {X 0,Y 367.972,Z 808.867,A -85,B 0,C 180,E1 -12809.774,E2 -12809.774} C_VEL
LIN {X 0,Y 367.728,Z 810.73,A -85,B 0,C 180,E1 -12811.066,E2 -12811.066} C_VEL
LIN {X 0,Y 367.51,Z 812.248,A -85,B 0,C 180,E1 -12812.712,E2 -12812.712} C_VEL
LIN {X 0,Y 367.414,Z 812.871,A -85,B 0,C 180,E1 -12814.665,E2 -12814.665} C_VEL
LIN {X 0,Y 367.424,Z 812.232,A -85,B 0,C 180,E1 -12816.55,E2 -12816.55} C_VEL
LIN {X 0,Y 367.546,Z 810.444,A -85,B 0,C 180,E1 -12818.376,E2 -12818.376} C_VEL
LIN {X 0,Y 367.883,Z 806.864,A -85,B 0,C 180,E1 -12820.506,E2 -12820.506} C_VEL
LIN {X 0,Y 368.163,Z 802.545,A -85,B 0,C 180,E1 -12822.291,E2 -12822.291} C_VEL
LIN {X 0,Y 368.673,Z 796.566,A -85,B 0,C 180,E1 -12824.142,E2 -12824.142} C_VEL
LIN {X 0,Y 369.24,Z 790.166,A -85,B 0,C 180,E1 -12825.708,E2 -12825.708} C_VEL
LIN {X 0,Y 369.944,Z 782.398,A -85,B 0,C 180,E1 -12827.249,E2 -12827.249} C_VEL
LIN {X 0,Y 370.715,Z 774.467,A -85,B 0,C 180,E1 -12828.54,E2 -12828.54} C_VEL
LIN {X 0,Y 371.624,Z 764.519,A -85,B 0,C 180,E1 -12829.871,E2 -12829.871} C_VEL
LIN {X 0,Y 372.522,Z 752.583,A -85,B 0,C 180,E1 -12831.137,E2 -12831.137} C_VEL
LIN {X 0,Y 373.387,Z 740.722,A -85,B 0,C 180,E1 -12832.122,E2 -12832.122} C_VEL
LIN {X 0,Y 374.05,Z 728.484,A -85,B 0,C 180,E1 -12832.889,E2 -12832.889} C_VEL
LIN {X 0,Y 374.542,Z 715.034,A -85,B 0,C 180,E1 -12833.494,E2 -12833.494} C_VEL
LIN {X 0,Y 374.928,Z 701.301,A -85,B 0,C 180,E1 -12833.869,E2 -12833.869} C_VEL
LIN {X 0,Y 376.325,Z 624.461,A -85,B 0,C 180,E1 -12835.483,E2 -12835.483} C_VEL
LIN {X 0,Y 374.335,Z 616.463,A -85,B 0,C 180,E1 -12835.761,E2 -12835.761} C_VEL
LIN {X 0,Y 369.505,Z 602.306,A -85,B 0,C 180,E1 -12836.363,E2 -12836.363} C_VEL
LIN {X 0,Y 368.972,Z 599.523,A -85,B 0,C 180,E1 -12837.187,E2 -12837.187} C_VEL
LIN {X 0,Y 368.943,Z 599.524,A -85,B 0,C 180,E1 -12841.194,E2 -12841.194} C_VEL
LIN {X 0,Y 368.997,Z 599.524,A -85,B 0,C 180,E1 -12844.021,E2 -12844.021} C_VEL
LIN {X 0,Y 368.935,Z 599.526,A -85,B 0,C 180,E1 -12847.607,E2 -12847.607} C_VEL
LIN {X 0,Y 368.988,Z 599.518,A -85,B 0,C 180,E1 -12851.109,E2 -12851.109} C_VEL
LIN {X 0,Y 368.998,Z 599.521,A -85,B 0,C 180,E1 -12854.537,E2 -12854.537} C_VEL
LIN {X 0,Y 369.013,Z 599.517,A -85,B 0,C 180,E1 -12857.908,E2 -12857.908} C_VEL
LIN {X 0,Y 369.229,Z 599.489,A -85,B 0,C 180,E1 -12861.801,E2 -12861.801} C_VEL
LIN {X 0,Y 369.145,Z 599.504,A -85,B 0,C 180,E1 -12864.539,E2 -12864.539} C_VEL
LIN {X 0,Y 369.32,Z 599.477,A -85,B 0,C 180,E1 -12867.82,E2 -12867.82} C_VEL
LIN {X 0,Y 369.455,Z 599.461,A -85,B 0,C 180,E1 -12870.012,E2 -12870.012} C_VEL
LIN {X 0,Y 369.32,Z 599.479,A -85,B 0,C 180,E1 -12872.182,E2 -12872.182} C_VEL
LIN {X 0,Y 369.037,Z 599.513,A -85,B 0,C 180,E1 -12874.775,E2 -12874.775} C_VEL
LIN {X 0,Y 368.455,Z 599.585,A -85,B 0,C 180,E1 -12875.688,E2 -12875.688} C_VEL
LIN {X 0,Y 365.633,Z 599.938,A -85,B 0,C 180,E1 -12877.172,E2 -12877.172} C_VEL
LIN {X 0,Y 363.186,Z 600.244,A -85,B 0,C 180,E1 -12878.372,E2 -12878.372} C_VEL
LIN {X 0,Y 362.124,Z 600.375,A -85,B 0,C 180,E1 -12879.301,E2 -12879.301} C_VEL
LIN {X 0,Y 362.034,Z 600.385,A -85,B 0,C 180,E1 -12879.616,E2 -12879.616} C_VEL
LIN {X 0,Y 362,Z 600.389,A -85,B 0,C 180,E1 -12883.9,E2 -12883.9} C_VEL
LIN {X 0,Y 361.97,Z 600.392,A -85,B 0,C 180,E1 -12887.94,E2 -12887.94} C_VEL
LIN {X 0,Y 361.895,Z 600.402,A -85,B 0,C 180,E1 -12891.654,E2 -12891.654} C_VEL
LIN {X 0,Y 361.932,Z 600.401,A -85,B 0,C 180,E1 -12895.291,E2 -12895.291} C_VEL
LIN {X 0,Y 361.912,Z 600.4,A -85,B 0,C 180,E1 -12897.78,E2 -12897.78} C_VEL
LIN {X 0,Y 361.841,Z 600.41,A -85,B 0,C 180,E1 -12901.63,E2 -12901.63} C_VEL
LIN {X 0,Y 361.878,Z 600.409,A -85,B 0,C 180,E1 -12905.346,E2 -12905.346} C_VEL
LIN {X 0,Y 361.874,Z 600.409,A -85,B 0,C 180,E1 -12909.028,E2 -12909.028} C_VEL
LIN {X 0,Y 361.84,Z 600.41,A -85,B 0,C 180,E1 -12912.829,E2 -12912.829} C_VEL
LIN {X 0,Y 361.839,Z 600.41,A -85,B 0,C 180,E1 -12915.945,E2 -12915.945} C_VEL
LIN {X 0,Y 361.84,Z 600.413,A -85,B 0,C 180,E1 -12919.245,E2 -12919.245} C_VEL
LIN {X 0,Y 361.867,Z 600.406,A -85,B 0,C 180,E1 -12922.778,E2 -12922.778} C_VEL
LIN {X 0,Y 361.859,Z 600.411,A -85,B 0,C 180,E1 -12925.72,E2 -12925.72} C_VEL
LIN {X 0,Y 361.879,Z 600.41,A -85,B 0,C 180,E1 -12929.673,E2 -12929.673} C_VEL
LIN {X 0,Y 361.96,Z 600.398,A -85,B 0,C 180,E1 -12933.476,E2 -12933.476} C_VEL
LIN {X 0,Y 361.885,Z 600.404,A -85,B 0,C 180,E1 -12937.144,E2 -12937.144} C_VEL
LIN {X 0,Y 361.917,Z 600.399,A -85,B 0,C 180,E1 -12940.724,E2 -12940.724} C_VEL
LIN {X 0,Y 361.938,Z 600.397,A -85,B 0,C 180,E1 -12943.066,E2 -12943.066} C_VEL
LIN {X 0,Y 362.004,Z 600.389,A -85,B 0,C 180,E1 -12946.528,E2 -12946.528} C_VEL
LIN {X 0,Y 362.037,Z 600.39,A -85,B 0,C 180,E1 -12949.938,E2 -12949.938} C_VEL
LIN {X 0,Y 362.167,Z 600.368,A -85,B 0,C 180,E1 -12953.314,E2 -12953.314} C_VEL
LIN {X 0,Y 362.286,Z 600.356,A -85,B 0,C 180,E1 -12957.777,E2 -12957.777} C_VEL
LIN {X 0,Y 362.432,Z 600.339,A -85,B 0,C 180,E1 -12960,E2 -12960} C_VEL
LIN {X 0,Y 362.286,Z 600.36,A -85,B 0,C 180,E1 -12962.224,E2 -12962.224} C_VEL
LIN {X 0,Y 362.169,Z 600.37,A -85,B 0,C 180,E1 -12966.686,E2 -12966.686} C_VEL
LIN {X 0,Y 362.037,Z 600.387,A -85,B 0,C 180,E1 -12970.062,E2 -12970.062} C_VEL
LIN {X 0,Y 362.004,Z 600.39,A -85,B 0,C 180,E1 -12973.899,E2 -12973.899} C_VEL
LIN {X 0,Y 361.934,Z 600.399,A -85,B 0,C 180,E1 -12976.934,E2 -12976.934} C_VEL
LIN {X 0,Y 361.892,Z 600.408,A -85,B 0,C 180,E1 -12980.461,E2 -12980.461} C_VEL
LIN {X 0,Y 361.899,Z 600.403,A -85,B 0,C 180,E1 -12984.113,E2 -12984.113} C_VEL
LIN {X 0,Y 361.948,Z 600.402,A -85,B 0,C 180,E1 -12986.721,E2 -12986.721} C_VEL
LIN {X 0,Y 361.88,Z 600.406,A -85,B 0,C 180,E1 -12990.328,E2 -12990.328} C_VEL
LIN {X 0,Y 361.86,Z 600.408,A -85,B 0,C 180,E1 -12994.28,E2 -12994.28} C_VEL
LIN {X 0,Y 361.869,Z 600.408,A -85,B 0,C 180,E1 -12997.222,E2 -12997.222} C_VEL
LIN {X 0,Y 361.841,Z 600.413,A -85,B 0,C 180,E1 -13000.755,E2 -13000.755} C_VEL
LIN {X 0,Y 361.839,Z 600.41,A -85,B 0,C 180,E1 -13004.365,E2 -13004.365} C_VEL
LIN {X 0,Y 361.841,Z 600.41,A -85,B 0,C 180,E1 -13007.568,E2 -13007.568} C_VEL
LIN {X 0,Y 361.875,Z 600.409,A -85,B 0,C 180,E1 -13010.973,E2 -13010.973} C_VEL
LIN {X 0,Y 361.879,Z 600.405,A -85,B 0,C 180,E1 -13014.655,E2 -13014.655} C_VEL
LIN {X 0,Y 361.843,Z 600.412,A -85,B 0,C 180,E1 -13018.37,E2 -13018.37} C_VEL
LIN {X 0,Y 361.903,Z 600.602,A -85,B 0,C 180,E1 -13018.818,E2 -13018.818} C_VEL
LIN {X 0,Y 364.589,Z 612.901,A -85,B 0,C 180,E1 -13021.817,E2 -13021.817} C_VEL
LIN {X 0,Y 366.191,Z 621.358,A -85,B 0,C 180,E1 -13023.804,E2 -13023.804} C_VEL
LIN {X 0,Y 365.066,Z 633.677,A -85,B 0,C 180,E1 -13026.454,E2 -13026.454} C_VEL
LIN {X 0,Y 364.285,Z 642.709,A -85,B 0,C 180,E1 -13028.374,E2 -13028.374} C_VEL
LIN {X 0,Y 369.034,Z 678.835,A -85,B 0,C 180,E1 -13029.443,E2 -13029.443} C_VEL
LIN {X 0,Y 367.578,Z 751.724,A -85,B 0,C 180,E1 -13031.031,E2 -13031.031} C_VEL
LIN {X 0,Y 366.974,Z 765.235,A -85,B 0,C 180,E1 -13031.542,E2 -13031.542} C_VEL
LIN {X 0,Y 366.078,Z 778.12,A -85,B 0,C 180,E1 -13032.255,E2 -13032.255} C_VEL
LIN {X 0,Y 365.123,Z 790.73,A -85,B 0,C 180,E1 -13033.217,E2 -13033.217} C_VEL
LIN {X 0,Y 364.194,Z 800.706,A -85,B 0,C 180,E1 -13034.181,E2 -13034.181} C_VEL
LIN {X 0,Y 363.335,Z 811.181,A -85,B 0,C 180,E1 -13035.435,E2 -13035.435} C_VEL
LIN {X 0,Y 362.425,Z 820.569,A -85,B 0,C 180,E1 -13036.828,E2 -13036.828} C_VEL
LIN {X 0,Y 361.757,Z 828.307,A -85,B 0,C 180,E1 -13038.229,E2 -13038.229} C_VEL
LIN {X 0,Y 361.138,Z 835.88,A -85,B 0,C 180,E1 -13039.912,E2 -13039.912} C_VEL
